// TIA Portal V20 export
FUNCTION_BLOCK "LER_AlignCalibration"   // FB100, LAD
// stored: Access Published, MemoryReserve 100, SetENOAutomatically false
   VAR_INPUT
      enable : Bool;
      Anode : Bool;
      Cathode : Bool;
      AxisXHomePos { ExternalAccessible := 'False'; ExternalVisible := 'False'; ExternalWritable := 'False'} : LReal;
      AxisY1HomePos { ExternalAccessible := 'False'; ExternalVisible := 'False'; ExternalWritable := 'False'} : LReal;
      AxisY2HomePos { ExternalAccessible := 'False'; ExternalVisible := 'False'; ExternalWritable := 'False'} : LReal;
   END_VAR
   VAR_OUTPUT
      Visiontrigger : Bool;
      error : Bool;
      busy : Bool;
      done : Bool;
      status : Word;
   END_VAR
   VAR_IN_OUT
      moduleInterface : "LER_typeAlignCalibrationInterface";
      AlignTableAxisX : DB_ANY;
      AlignTableAxisY1 : DB_ANY;
      AlignTableAxisY2 : DB_ANY;
   END_VAR
   VAR
      statAxisXMovePosition : Array[1..9] of LReal;
      statAxisY1MovePosition : Array[1..9] of LReal;
      statAxisY2MovePosition : Array[1..9] of LReal;
      instAlignTableAxisXMCMoveAbs : MC_MOVEABSOLUTE;
      instAlignTableAxisY1MCMoveAbs { S7_SetPoint := 'True'} : MC_MOVEABSOLUTE;
      instAlignTableAxisY2MCMoveAbs { S7_SetPoint := 'True'} : MC_MOVEABSOLUTE;
      statPulse { S7_SetPoint := 'True'} : Array[1..50] of Bool;
      statMoveXCmd : Array[1..10] of Bool;
      statMoveY1Cmd : Array[1..10] of Bool;
      statMoveY2Cmd : Array[1..10] of Bool;
      statVisionCmd : Array[1..10] of Bool;
      statTimer : Array[1..20] of TON_TIME;
      statAllMoveSeq : DInt;
      statManualMove : Bool;
   END_VAR
   VAR_TEMP
      tempAlignTableAxisX : REF_TO TO_SynchronousAxis;
      tempAlignTableAxisY1 : REF_TO TO_SynchronousAxis;
      tempAlignTableAxisY2 : REF_TO TO_SynchronousAxis;
   END_VAR
   VAR CONSTANT
      VISION_DELAY_TIME : Time := T#500ms;
   END_VAR
   VAR_TEMP   // added for the SCL form of the ladder/FBD networks
      _w1 : Bool;
      _w2 : Bool;
   END_VAR
BEGIN

REGION Network 1 (SCL): Axis Config
   #tempAlignTableAxisX ?= #AlignTableAxisX;
   #tempAlignTableAxisY1 ?= #AlignTableAxisY1;
   #tempAlignTableAxisY2 ?= #AlignTableAxisY2;
END_REGION

REGION Network 2: Standard Postion Config
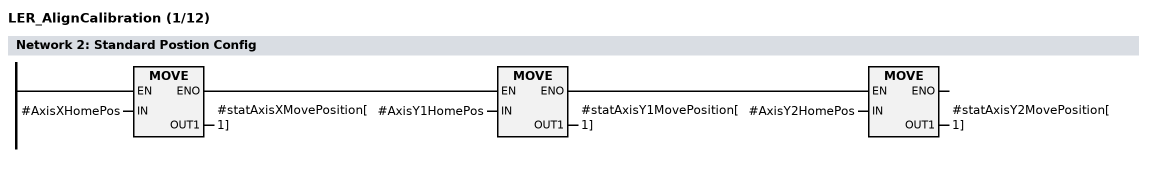
   RUNG wire#powerrail
      Move(in := #AxisXHomePos, out1 => #statAxisXMovePosition[1])
      Move(in := #AxisY1HomePos, out1 => #statAxisY1MovePosition[1])
      Move(in := #AxisY2HomePos, out1 => #statAxisY2MovePosition[1])
   END_RUNG
   // the same network as SCL:
   #statAxisXMovePosition[1] := #AxisXHomePos;
   #statAxisY1MovePosition[1] := #AxisY1HomePos;
   #statAxisY2MovePosition[1] := #AxisY2HomePos;
END_REGION

REGION Network 3: Anode MovePosition Config
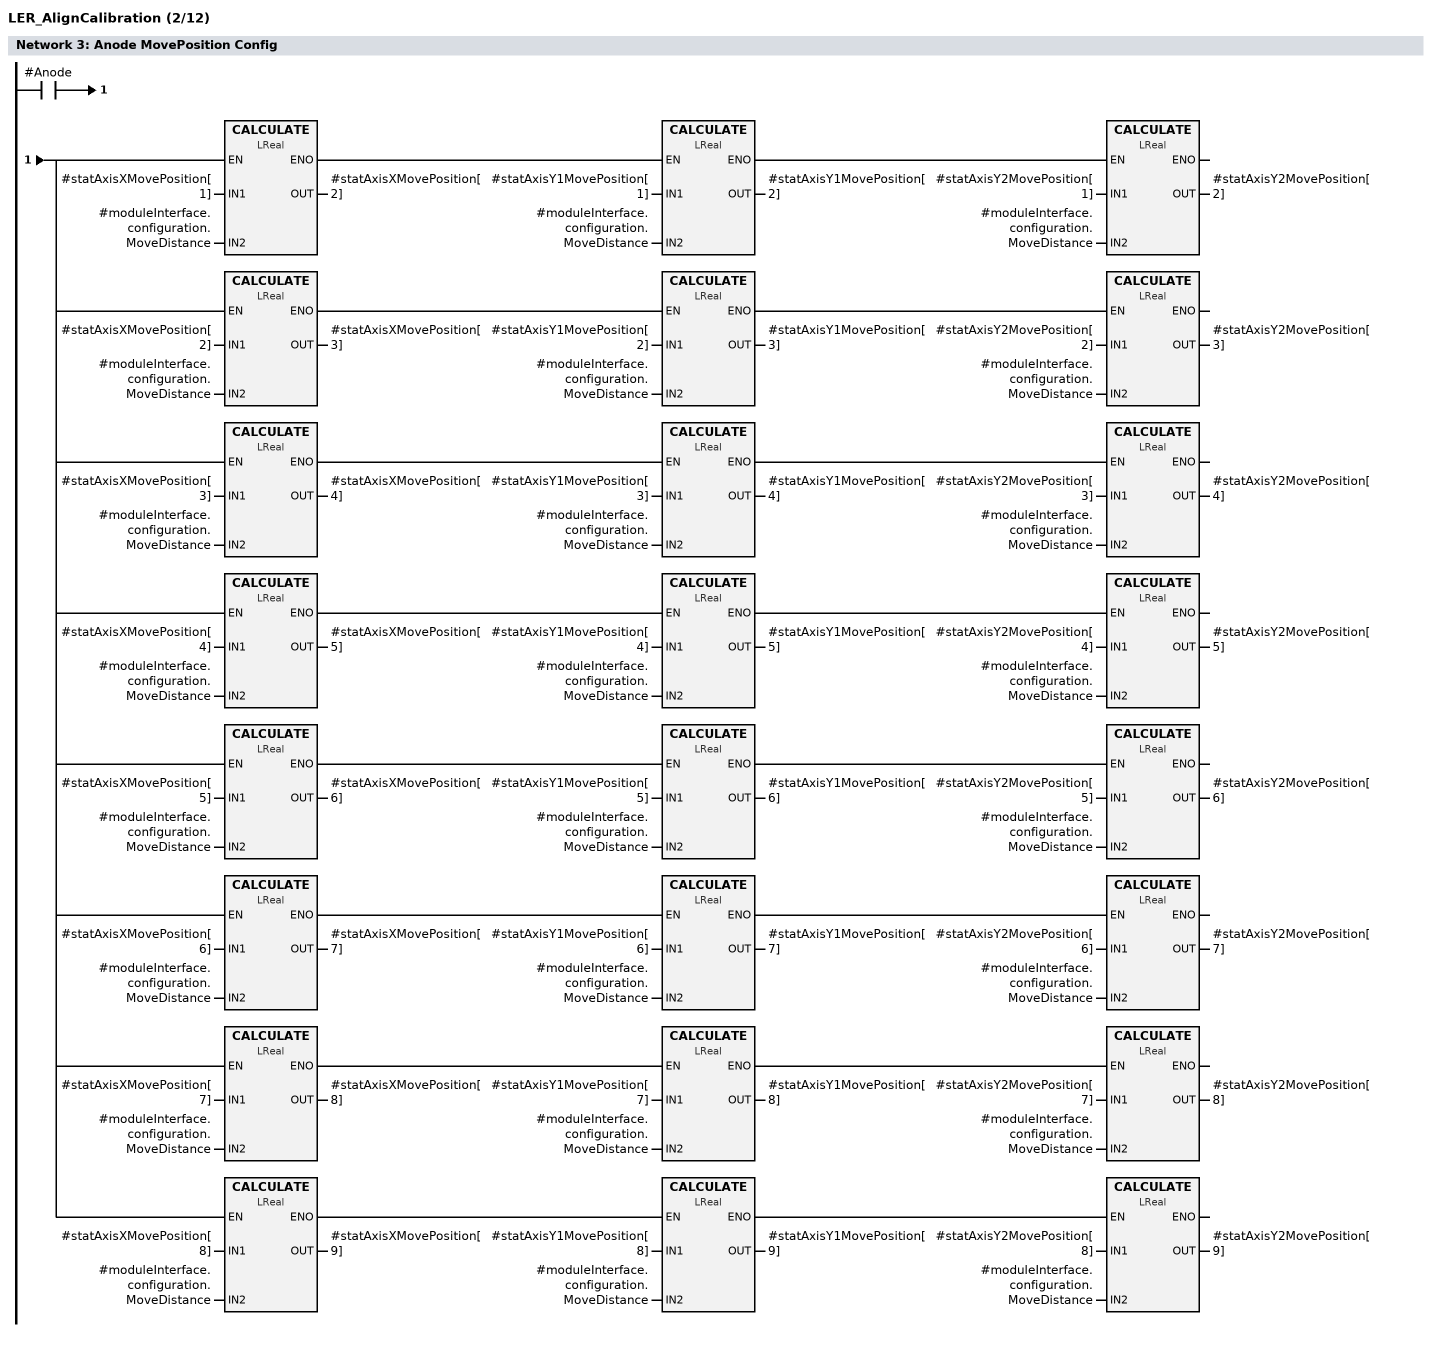
   RUNG wire#powerrail
      Contact( #Anode )
      wire#w1
      { S7_Templates := "SrcType := LReal"; S7_Expression := "IN1-IN2" } Calculate(in1 := #statAxisXMovePosition[1], in2 := #moduleInterface.configuration.MoveDistance, out => #statAxisXMovePosition[2])
      { S7_Templates := "SrcType := LReal"; S7_Expression := "IN1" } Calculate(in1 := #statAxisY1MovePosition[1], in2 := #moduleInterface.configuration.MoveDistance, out => #statAxisY1MovePosition[2])
      { S7_Templates := "SrcType := LReal"; S7_Expression := "IN1" } Calculate(in1 := #statAxisY2MovePosition[1], in2 := #moduleInterface.configuration.MoveDistance, out => #statAxisY2MovePosition[2])
   END_RUNG
   RUNG wire#w1
      { S7_Templates := "SrcType := LReal"; S7_Expression := "IN1" } Calculate(in1 := #statAxisXMovePosition[2], in2 := #moduleInterface.configuration.MoveDistance, out => #statAxisXMovePosition[3])
      { S7_Templates := "SrcType := LReal"; S7_Expression := "IN1+IN2" } Calculate(in1 := #statAxisY1MovePosition[2], in2 := #moduleInterface.configuration.MoveDistance, out => #statAxisY1MovePosition[3])
      { S7_Templates := "SrcType := LReal"; S7_Expression := "IN1-IN2" } Calculate(in1 := #statAxisY2MovePosition[2], in2 := #moduleInterface.configuration.MoveDistance, out => #statAxisY2MovePosition[3])
   END_RUNG
   RUNG wire#w1
      { S7_Templates := "SrcType := LReal"; S7_Expression := "IN1+IN2" } Calculate(in1 := #statAxisXMovePosition[3], in2 := #moduleInterface.configuration.MoveDistance, out => #statAxisXMovePosition[4])
      { S7_Templates := "SrcType := LReal"; S7_Expression := "IN1" } Calculate(in1 := #statAxisY1MovePosition[3], in2 := #moduleInterface.configuration.MoveDistance, out => #statAxisY1MovePosition[4])
      { S7_Templates := "SrcType := LReal"; S7_Expression := "IN1" } Calculate(in1 := #statAxisY2MovePosition[3], in2 := #moduleInterface.configuration.MoveDistance, out => #statAxisY2MovePosition[4])
   END_RUNG
   RUNG wire#w1
      { S7_Templates := "SrcType := LReal"; S7_Expression := "IN1+IN2" } Calculate(in1 := #statAxisXMovePosition[4], in2 := #moduleInterface.configuration.MoveDistance, out => #statAxisXMovePosition[5])
      { S7_Templates := "SrcType := LReal"; S7_Expression := "IN1" } Calculate(in1 := #statAxisY1MovePosition[4], in2 := #moduleInterface.configuration.MoveDistance, out => #statAxisY1MovePosition[5])
      { S7_Templates := "SrcType := LReal"; S7_Expression := "IN1" } Calculate(in1 := #statAxisY2MovePosition[4], in2 := #moduleInterface.configuration.MoveDistance, out => #statAxisY2MovePosition[5])
   END_RUNG
   RUNG wire#w1
      { S7_Templates := "SrcType := LReal"; S7_Expression := "IN1" } Calculate(in1 := #statAxisXMovePosition[5], in2 := #moduleInterface.configuration.MoveDistance, out => #statAxisXMovePosition[6])
      { S7_Templates := "SrcType := LReal"; S7_Expression := "IN1-IN2" } Calculate(in1 := #statAxisY1MovePosition[5], in2 := #moduleInterface.configuration.MoveDistance, out => #statAxisY1MovePosition[6])
      { S7_Templates := "SrcType := LReal"; S7_Expression := "IN1+IN2" } Calculate(in1 := #statAxisY2MovePosition[5], in2 := #moduleInterface.configuration.MoveDistance, out => #statAxisY2MovePosition[6])
   END_RUNG
   RUNG wire#w1
      { S7_Templates := "SrcType := LReal"; S7_Expression := "IN1" } Calculate(in1 := #statAxisXMovePosition[6], in2 := #moduleInterface.configuration.MoveDistance, out => #statAxisXMovePosition[7])
      { S7_Templates := "SrcType := LReal"; S7_Expression := "IN1-IN2" } Calculate(in1 := #statAxisY1MovePosition[6], in2 := #moduleInterface.configuration.MoveDistance, out => #statAxisY1MovePosition[7])
      { S7_Templates := "SrcType := LReal"; S7_Expression := "IN1+IN2" } Calculate(in1 := #statAxisY2MovePosition[6], in2 := #moduleInterface.configuration.MoveDistance, out => #statAxisY2MovePosition[7])
   END_RUNG
   RUNG wire#w1
      { S7_Templates := "SrcType := LReal"; S7_Expression := "IN1-IN2" } Calculate(in1 := #statAxisXMovePosition[7], in2 := #moduleInterface.configuration.MoveDistance, out => #statAxisXMovePosition[8])
      { S7_Templates := "SrcType := LReal"; S7_Expression := "IN1" } Calculate(in1 := #statAxisY1MovePosition[7], in2 := #moduleInterface.configuration.MoveDistance, out => #statAxisY1MovePosition[8])
      { S7_Templates := "SrcType := LReal"; S7_Expression := "IN1" } Calculate(in1 := #statAxisY2MovePosition[7], in2 := #moduleInterface.configuration.MoveDistance, out => #statAxisY2MovePosition[8])
   END_RUNG
   RUNG wire#w1
      { S7_Templates := "SrcType := LReal"; S7_Expression := "IN1-IN2" } Calculate(in1 := #statAxisXMovePosition[8], in2 := #moduleInterface.configuration.MoveDistance, out => #statAxisXMovePosition[9])
      { S7_Templates := "SrcType := LReal"; S7_Expression := "IN1" } Calculate(in1 := #statAxisY1MovePosition[8], in2 := #moduleInterface.configuration.MoveDistance, out => #statAxisY1MovePosition[9])
      { S7_Templates := "SrcType := LReal"; S7_Expression := "IN1" } Calculate(in1 := #statAxisY2MovePosition[8], in2 := #moduleInterface.configuration.MoveDistance, out => #statAxisY2MovePosition[9])
   END_RUNG
   // the same network as SCL:
   IF #Anode THEN
       #statAxisXMovePosition[2] := #statAxisXMovePosition[1]-#moduleInterface.configuration.MoveDistance;
       #statAxisY1MovePosition[2] := #statAxisY1MovePosition[1];
       #statAxisY2MovePosition[2] := #statAxisY2MovePosition[1];
       #statAxisXMovePosition[3] := #statAxisXMovePosition[2];
       #statAxisY1MovePosition[3] := #statAxisY1MovePosition[2]+#moduleInterface.configuration.MoveDistance;
       #statAxisY2MovePosition[3] := #statAxisY2MovePosition[2]-#moduleInterface.configuration.MoveDistance;
       #statAxisXMovePosition[4] := #statAxisXMovePosition[3]+#moduleInterface.configuration.MoveDistance;
       #statAxisY1MovePosition[4] := #statAxisY1MovePosition[3];
       #statAxisY2MovePosition[4] := #statAxisY2MovePosition[3];
       #statAxisXMovePosition[5] := #statAxisXMovePosition[4]+#moduleInterface.configuration.MoveDistance;
       #statAxisY1MovePosition[5] := #statAxisY1MovePosition[4];
       #statAxisY2MovePosition[5] := #statAxisY2MovePosition[4];
       #statAxisXMovePosition[6] := #statAxisXMovePosition[5];
       #statAxisY1MovePosition[6] := #statAxisY1MovePosition[5]-#moduleInterface.configuration.MoveDistance;
       #statAxisY2MovePosition[6] := #statAxisY2MovePosition[5]+#moduleInterface.configuration.MoveDistance;
       #statAxisXMovePosition[7] := #statAxisXMovePosition[6];
       #statAxisY1MovePosition[7] := #statAxisY1MovePosition[6]-#moduleInterface.configuration.MoveDistance;
       #statAxisY2MovePosition[7] := #statAxisY2MovePosition[6]+#moduleInterface.configuration.MoveDistance;
       #statAxisXMovePosition[8] := #statAxisXMovePosition[7]-#moduleInterface.configuration.MoveDistance;
       #statAxisY1MovePosition[8] := #statAxisY1MovePosition[7];
       #statAxisY2MovePosition[8] := #statAxisY2MovePosition[7];
       #statAxisXMovePosition[9] := #statAxisXMovePosition[8]-#moduleInterface.configuration.MoveDistance;
       #statAxisY1MovePosition[9] := #statAxisY1MovePosition[8];
       #statAxisY2MovePosition[9] := #statAxisY2MovePosition[8];
   END_IF;
END_REGION

REGION Network 4: Cathode MovePosition Config
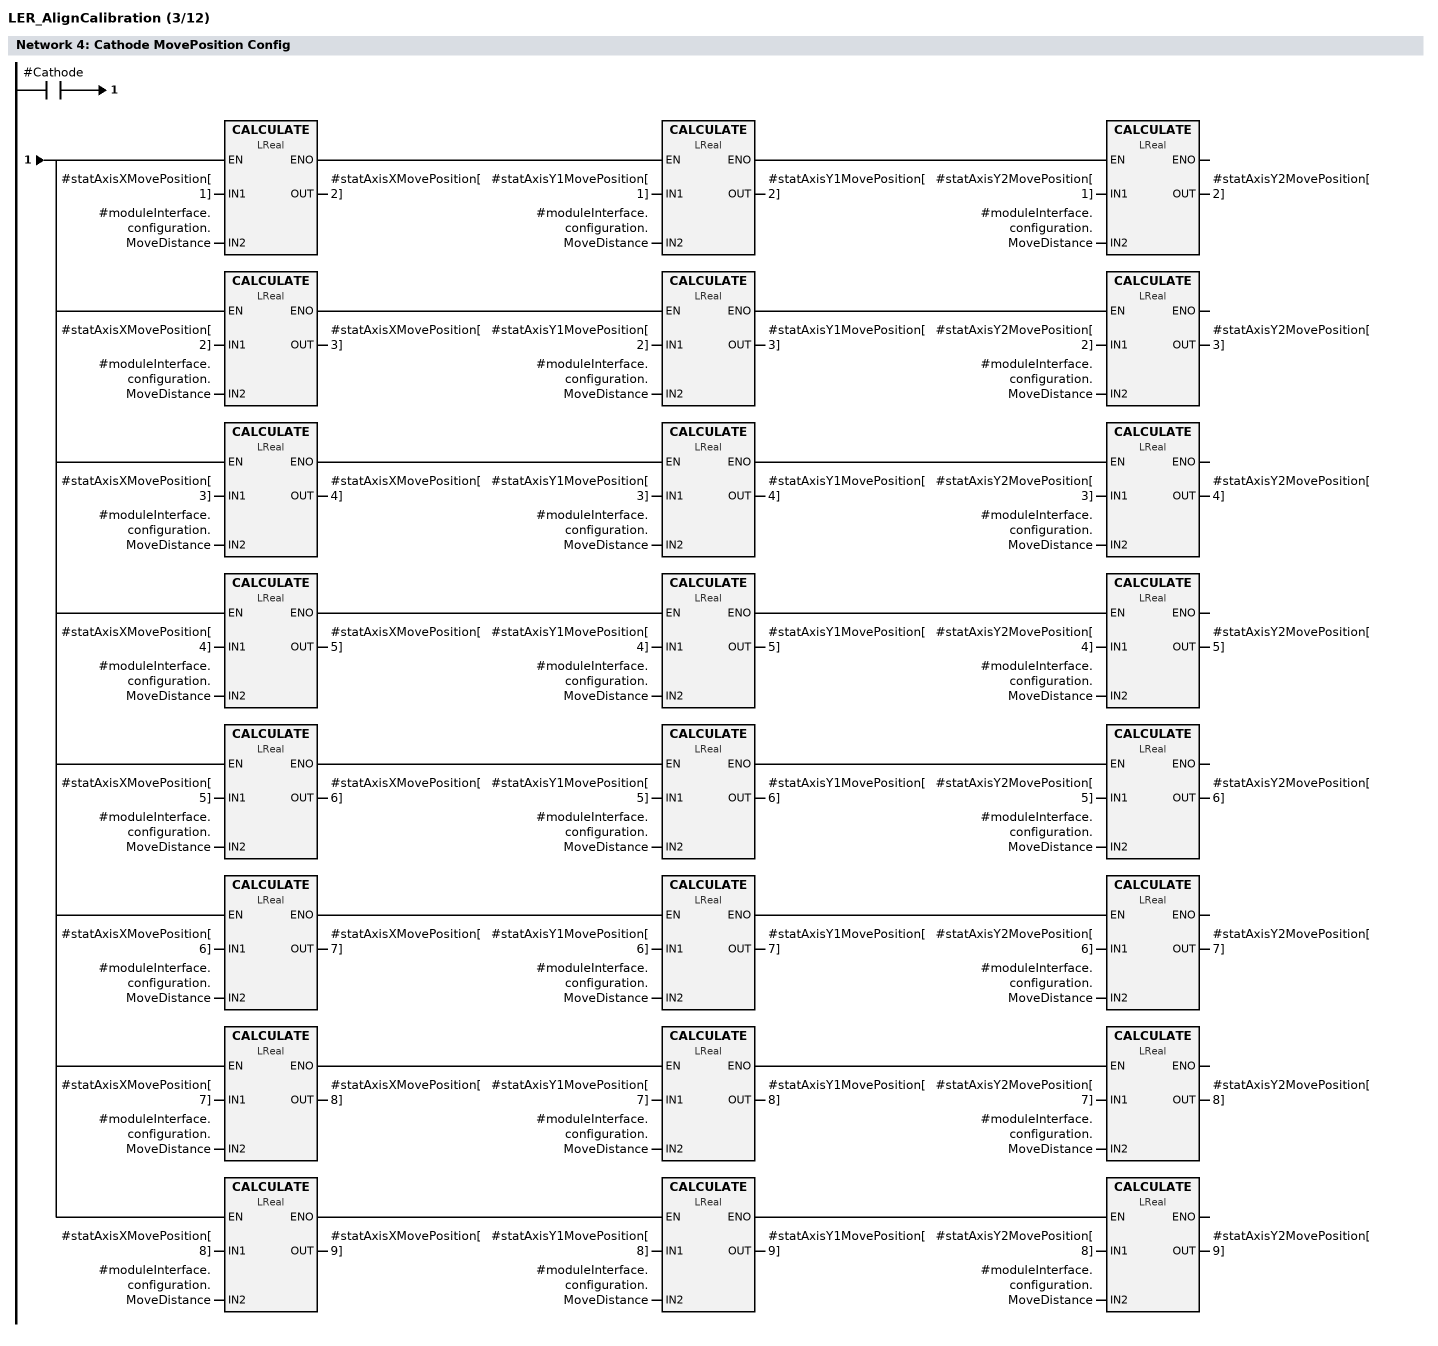
   RUNG wire#powerrail
      Contact( #Cathode )
      wire#w1
      { S7_Templates := "SrcType := LReal"; S7_Expression := "IN1+IN2" } Calculate(in1 := #statAxisXMovePosition[1], in2 := #moduleInterface.configuration.MoveDistance, out => #statAxisXMovePosition[2])
      { S7_Templates := "SrcType := LReal"; S7_Expression := "IN1" } Calculate(in1 := #statAxisY1MovePosition[1], in2 := #moduleInterface.configuration.MoveDistance, out => #statAxisY1MovePosition[2])
      { S7_Templates := "SrcType := LReal"; S7_Expression := "IN1" } Calculate(in1 := #statAxisY2MovePosition[1], in2 := #moduleInterface.configuration.MoveDistance, out => #statAxisY2MovePosition[2])
   END_RUNG
   RUNG wire#w1
      { S7_Templates := "SrcType := LReal"; S7_Expression := "IN1" } Calculate(in1 := #statAxisXMovePosition[2], in2 := #moduleInterface.configuration.MoveDistance, out => #statAxisXMovePosition[3])
      { S7_Templates := "SrcType := LReal"; S7_Expression := "IN1+IN2" } Calculate(in1 := #statAxisY1MovePosition[2], in2 := #moduleInterface.configuration.MoveDistance, out => #statAxisY1MovePosition[3])
      { S7_Templates := "SrcType := LReal"; S7_Expression := "IN1-IN2" } Calculate(in1 := #statAxisY2MovePosition[2], in2 := #moduleInterface.configuration.MoveDistance, out => #statAxisY2MovePosition[3])
   END_RUNG
   RUNG wire#w1
      { S7_Templates := "SrcType := LReal"; S7_Expression := "IN1-IN2" } Calculate(in1 := #statAxisXMovePosition[3], in2 := #moduleInterface.configuration.MoveDistance, out => #statAxisXMovePosition[4])
      { S7_Templates := "SrcType := LReal"; S7_Expression := "IN1" } Calculate(in1 := #statAxisY1MovePosition[3], in2 := #moduleInterface.configuration.MoveDistance, out => #statAxisY1MovePosition[4])
      { S7_Templates := "SrcType := LReal"; S7_Expression := "IN1" } Calculate(in1 := #statAxisY2MovePosition[3], in2 := #moduleInterface.configuration.MoveDistance, out => #statAxisY2MovePosition[4])
   END_RUNG
   RUNG wire#w1
      { S7_Templates := "SrcType := LReal"; S7_Expression := "IN1-IN2" } Calculate(in1 := #statAxisXMovePosition[4], in2 := #moduleInterface.configuration.MoveDistance, out => #statAxisXMovePosition[5])
      { S7_Templates := "SrcType := LReal"; S7_Expression := "IN1" } Calculate(in1 := #statAxisY1MovePosition[4], in2 := #moduleInterface.configuration.MoveDistance, out => #statAxisY1MovePosition[5])
      { S7_Templates := "SrcType := LReal"; S7_Expression := "IN1" } Calculate(in1 := #statAxisY2MovePosition[4], in2 := #moduleInterface.configuration.MoveDistance, out => #statAxisY2MovePosition[5])
   END_RUNG
   RUNG wire#w1
      { S7_Templates := "SrcType := LReal"; S7_Expression := "IN1" } Calculate(in1 := #statAxisXMovePosition[5], in2 := #moduleInterface.configuration.MoveDistance, out => #statAxisXMovePosition[6])
      { S7_Templates := "SrcType := LReal"; S7_Expression := "IN1-IN2" } Calculate(in1 := #statAxisY1MovePosition[5], in2 := #moduleInterface.configuration.MoveDistance, out => #statAxisY1MovePosition[6])
      { S7_Templates := "SrcType := LReal"; S7_Expression := "IN1+IN2" } Calculate(in1 := #statAxisY2MovePosition[5], in2 := #moduleInterface.configuration.MoveDistance, out => #statAxisY2MovePosition[6])
   END_RUNG
   RUNG wire#w1
      { S7_Templates := "SrcType := LReal"; S7_Expression := "IN1" } Calculate(in1 := #statAxisXMovePosition[6], in2 := #moduleInterface.configuration.MoveDistance, out => #statAxisXMovePosition[7])
      { S7_Templates := "SrcType := LReal"; S7_Expression := "IN1-IN2" } Calculate(in1 := #statAxisY1MovePosition[6], in2 := #moduleInterface.configuration.MoveDistance, out => #statAxisY1MovePosition[7])
      { S7_Templates := "SrcType := LReal"; S7_Expression := "IN1+IN2" } Calculate(in1 := #statAxisY2MovePosition[6], in2 := #moduleInterface.configuration.MoveDistance, out => #statAxisY2MovePosition[7])
   END_RUNG
   RUNG wire#w1
      { S7_Templates := "SrcType := LReal"; S7_Expression := "IN1+IN2" } Calculate(in1 := #statAxisXMovePosition[7], in2 := #moduleInterface.configuration.MoveDistance, out => #statAxisXMovePosition[8])
      { S7_Templates := "SrcType := LReal"; S7_Expression := "IN1" } Calculate(in1 := #statAxisY1MovePosition[7], in2 := #moduleInterface.configuration.MoveDistance, out => #statAxisY1MovePosition[8])
      { S7_Templates := "SrcType := LReal"; S7_Expression := "IN1" } Calculate(in1 := #statAxisY2MovePosition[7], in2 := #moduleInterface.configuration.MoveDistance, out => #statAxisY2MovePosition[8])
   END_RUNG
   RUNG wire#w1
      { S7_Templates := "SrcType := LReal"; S7_Expression := "IN1+IN2" } Calculate(in1 := #statAxisXMovePosition[8], in2 := #moduleInterface.configuration.MoveDistance, out => #statAxisXMovePosition[9])
      { S7_Templates := "SrcType := LReal"; S7_Expression := "IN1" } Calculate(in1 := #statAxisY1MovePosition[8], in2 := #moduleInterface.configuration.MoveDistance, out => #statAxisY1MovePosition[9])
      { S7_Templates := "SrcType := LReal"; S7_Expression := "IN1" } Calculate(in1 := #statAxisY2MovePosition[8], in2 := #moduleInterface.configuration.MoveDistance, out => #statAxisY2MovePosition[9])
   END_RUNG
   // the same network as SCL:
   IF #Cathode THEN
       #statAxisXMovePosition[2] := #statAxisXMovePosition[1]+#moduleInterface.configuration.MoveDistance;
       #statAxisY1MovePosition[2] := #statAxisY1MovePosition[1];
       #statAxisY2MovePosition[2] := #statAxisY2MovePosition[1];
       #statAxisXMovePosition[3] := #statAxisXMovePosition[2];
       #statAxisY1MovePosition[3] := #statAxisY1MovePosition[2]+#moduleInterface.configuration.MoveDistance;
       #statAxisY2MovePosition[3] := #statAxisY2MovePosition[2]-#moduleInterface.configuration.MoveDistance;
       #statAxisXMovePosition[4] := #statAxisXMovePosition[3]-#moduleInterface.configuration.MoveDistance;
       #statAxisY1MovePosition[4] := #statAxisY1MovePosition[3];
       #statAxisY2MovePosition[4] := #statAxisY2MovePosition[3];
       #statAxisXMovePosition[5] := #statAxisXMovePosition[4]-#moduleInterface.configuration.MoveDistance;
       #statAxisY1MovePosition[5] := #statAxisY1MovePosition[4];
       #statAxisY2MovePosition[5] := #statAxisY2MovePosition[4];
       #statAxisXMovePosition[6] := #statAxisXMovePosition[5];
       #statAxisY1MovePosition[6] := #statAxisY1MovePosition[5]-#moduleInterface.configuration.MoveDistance;
       #statAxisY2MovePosition[6] := #statAxisY2MovePosition[5]+#moduleInterface.configuration.MoveDistance;
       #statAxisXMovePosition[7] := #statAxisXMovePosition[6];
       #statAxisY1MovePosition[7] := #statAxisY1MovePosition[6]-#moduleInterface.configuration.MoveDistance;
       #statAxisY2MovePosition[7] := #statAxisY2MovePosition[6]+#moduleInterface.configuration.MoveDistance;
       #statAxisXMovePosition[8] := #statAxisXMovePosition[7]+#moduleInterface.configuration.MoveDistance;
       #statAxisY1MovePosition[8] := #statAxisY1MovePosition[7];
       #statAxisY2MovePosition[8] := #statAxisY2MovePosition[7];
       #statAxisXMovePosition[9] := #statAxisXMovePosition[8]+#moduleInterface.configuration.MoveDistance;
       #statAxisY1MovePosition[9] := #statAxisY1MovePosition[8];
       #statAxisY2MovePosition[9] := #statAxisY2MovePosition[8];
   END_IF;
END_REGION

REGION Network 5: All Move Seq Start/Stop And Error Check
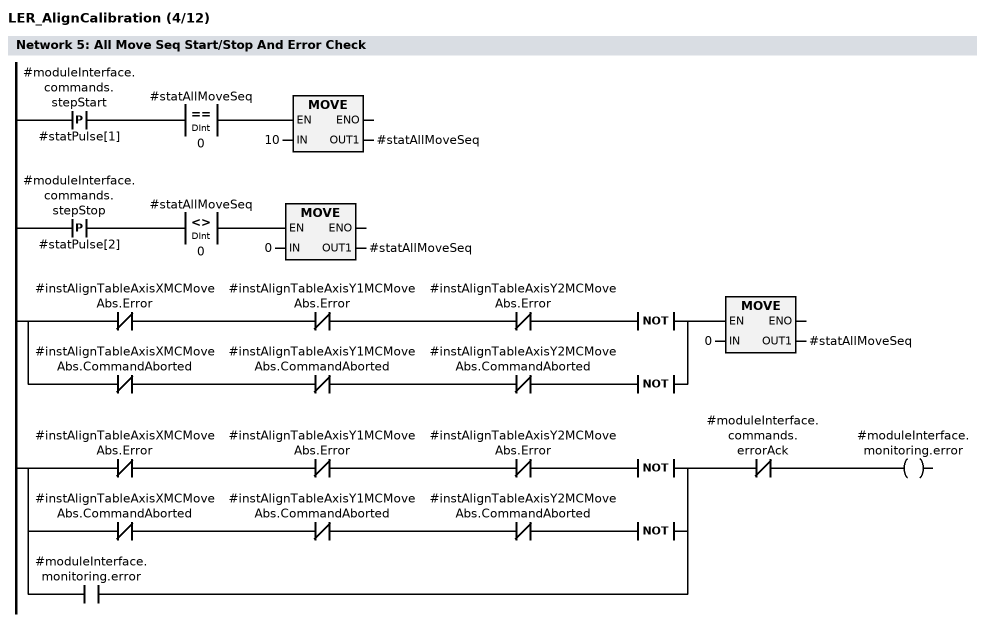
   RUNG wire#powerrail
      P_Contact(operand := #moduleInterface.commands.stepStart, bit := #statPulse[1])
      { S7_Templates := "SrcType := DInt" } EQ_Contact(in1 := #statAllMoveSeq, in2 := 0)
      Move(in := 10, out1 => #statAllMoveSeq)
   END_RUNG
   RUNG wire#powerrail
      P_Contact(operand := #moduleInterface.commands.stepStop, bit := #statPulse[2])
      { S7_Templates := "SrcType := DInt" } NE_Contact(in1 := #statAllMoveSeq, in2 := 0)
      Move(in := 0, out1 => #statAllMoveSeq)
   END_RUNG
   RUNG wire#powerrail
      I_Contact( #instAlignTableAxisXMCMoveAbs.Error )
      I_Contact( #instAlignTableAxisY1MCMoveAbs.Error )
      I_Contact( #instAlignTableAxisY2MCMoveAbs.Error )
      Not()
      wire#w1
      Move(in := 0, out1 => #statAllMoveSeq)
   END_RUNG
   RUNG wire#powerrail
      I_Contact( #instAlignTableAxisXMCMoveAbs.CommandAborted )
      I_Contact( #instAlignTableAxisY1MCMoveAbs.CommandAborted )
      I_Contact( #instAlignTableAxisY2MCMoveAbs.CommandAborted )
      Not()
   END_RUNG wire#w1
   RUNG wire#powerrail
      I_Contact( #instAlignTableAxisXMCMoveAbs.Error )
      I_Contact( #instAlignTableAxisY1MCMoveAbs.Error )
      I_Contact( #instAlignTableAxisY2MCMoveAbs.Error )
      Not()
      wire#w2
      I_Contact( #moduleInterface.commands.errorAck )
      Coil( #moduleInterface.monitoring.error )
   END_RUNG
   RUNG wire#powerrail
      I_Contact( #instAlignTableAxisXMCMoveAbs.CommandAborted )
      I_Contact( #instAlignTableAxisY1MCMoveAbs.CommandAborted )
      I_Contact( #instAlignTableAxisY2MCMoveAbs.CommandAborted )
      Not()
   END_RUNG wire#w2
   RUNG wire#powerrail
      Contact( #moduleInterface.monitoring.error )
   END_RUNG wire#w2
   // the same network as SCL:
   #_w1 := #moduleInterface.commands.stepStart AND NOT #statPulse[1];   // rising edge of #moduleInterface.commands.stepStart
   #statPulse[1] := #moduleInterface.commands.stepStart;
   IF #_w1 AND (#statAllMoveSeq = 0) THEN #statAllMoveSeq := 10; END_IF;
   #_w2 := #moduleInterface.commands.stepStop AND NOT #statPulse[2];   // rising edge of #moduleInterface.commands.stepStop
   #statPulse[2] := #moduleInterface.commands.stepStop;
   IF #_w2 AND (#statAllMoveSeq <> 0) THEN #statAllMoveSeq := 0; END_IF;
   IF NOT (NOT #instAlignTableAxisXMCMoveAbs.Error AND NOT #instAlignTableAxisY1MCMoveAbs.Error AND NOT #instAlignTableAxisY2MCMoveAbs.Error) OR NOT (NOT #instAlignTableAxisXMCMoveAbs.CommandAborted AND NOT #instAlignTableAxisY1MCMoveAbs.CommandAborted AND NOT #instAlignTableAxisY2MCMoveAbs.CommandAborted) THEN
       #statAllMoveSeq := 0;
   END_IF;
   #moduleInterface.monitoring.error := (NOT (NOT #instAlignTableAxisXMCMoveAbs.Error AND NOT #instAlignTableAxisY1MCMoveAbs.Error AND NOT #instAlignTableAxisY2MCMoveAbs.Error) OR NOT (NOT #instAlignTableAxisXMCMoveAbs.CommandAborted AND NOT #instAlignTableAxisY1MCMoveAbs.CommandAborted AND NOT #instAlignTableAxisY2MCMoveAbs.CommandAborted) OR #moduleInterface.monitoring.error) AND NOT #moduleInterface.commands.errorAck;
END_REGION

REGION Network 6: Manual Move Pos Check
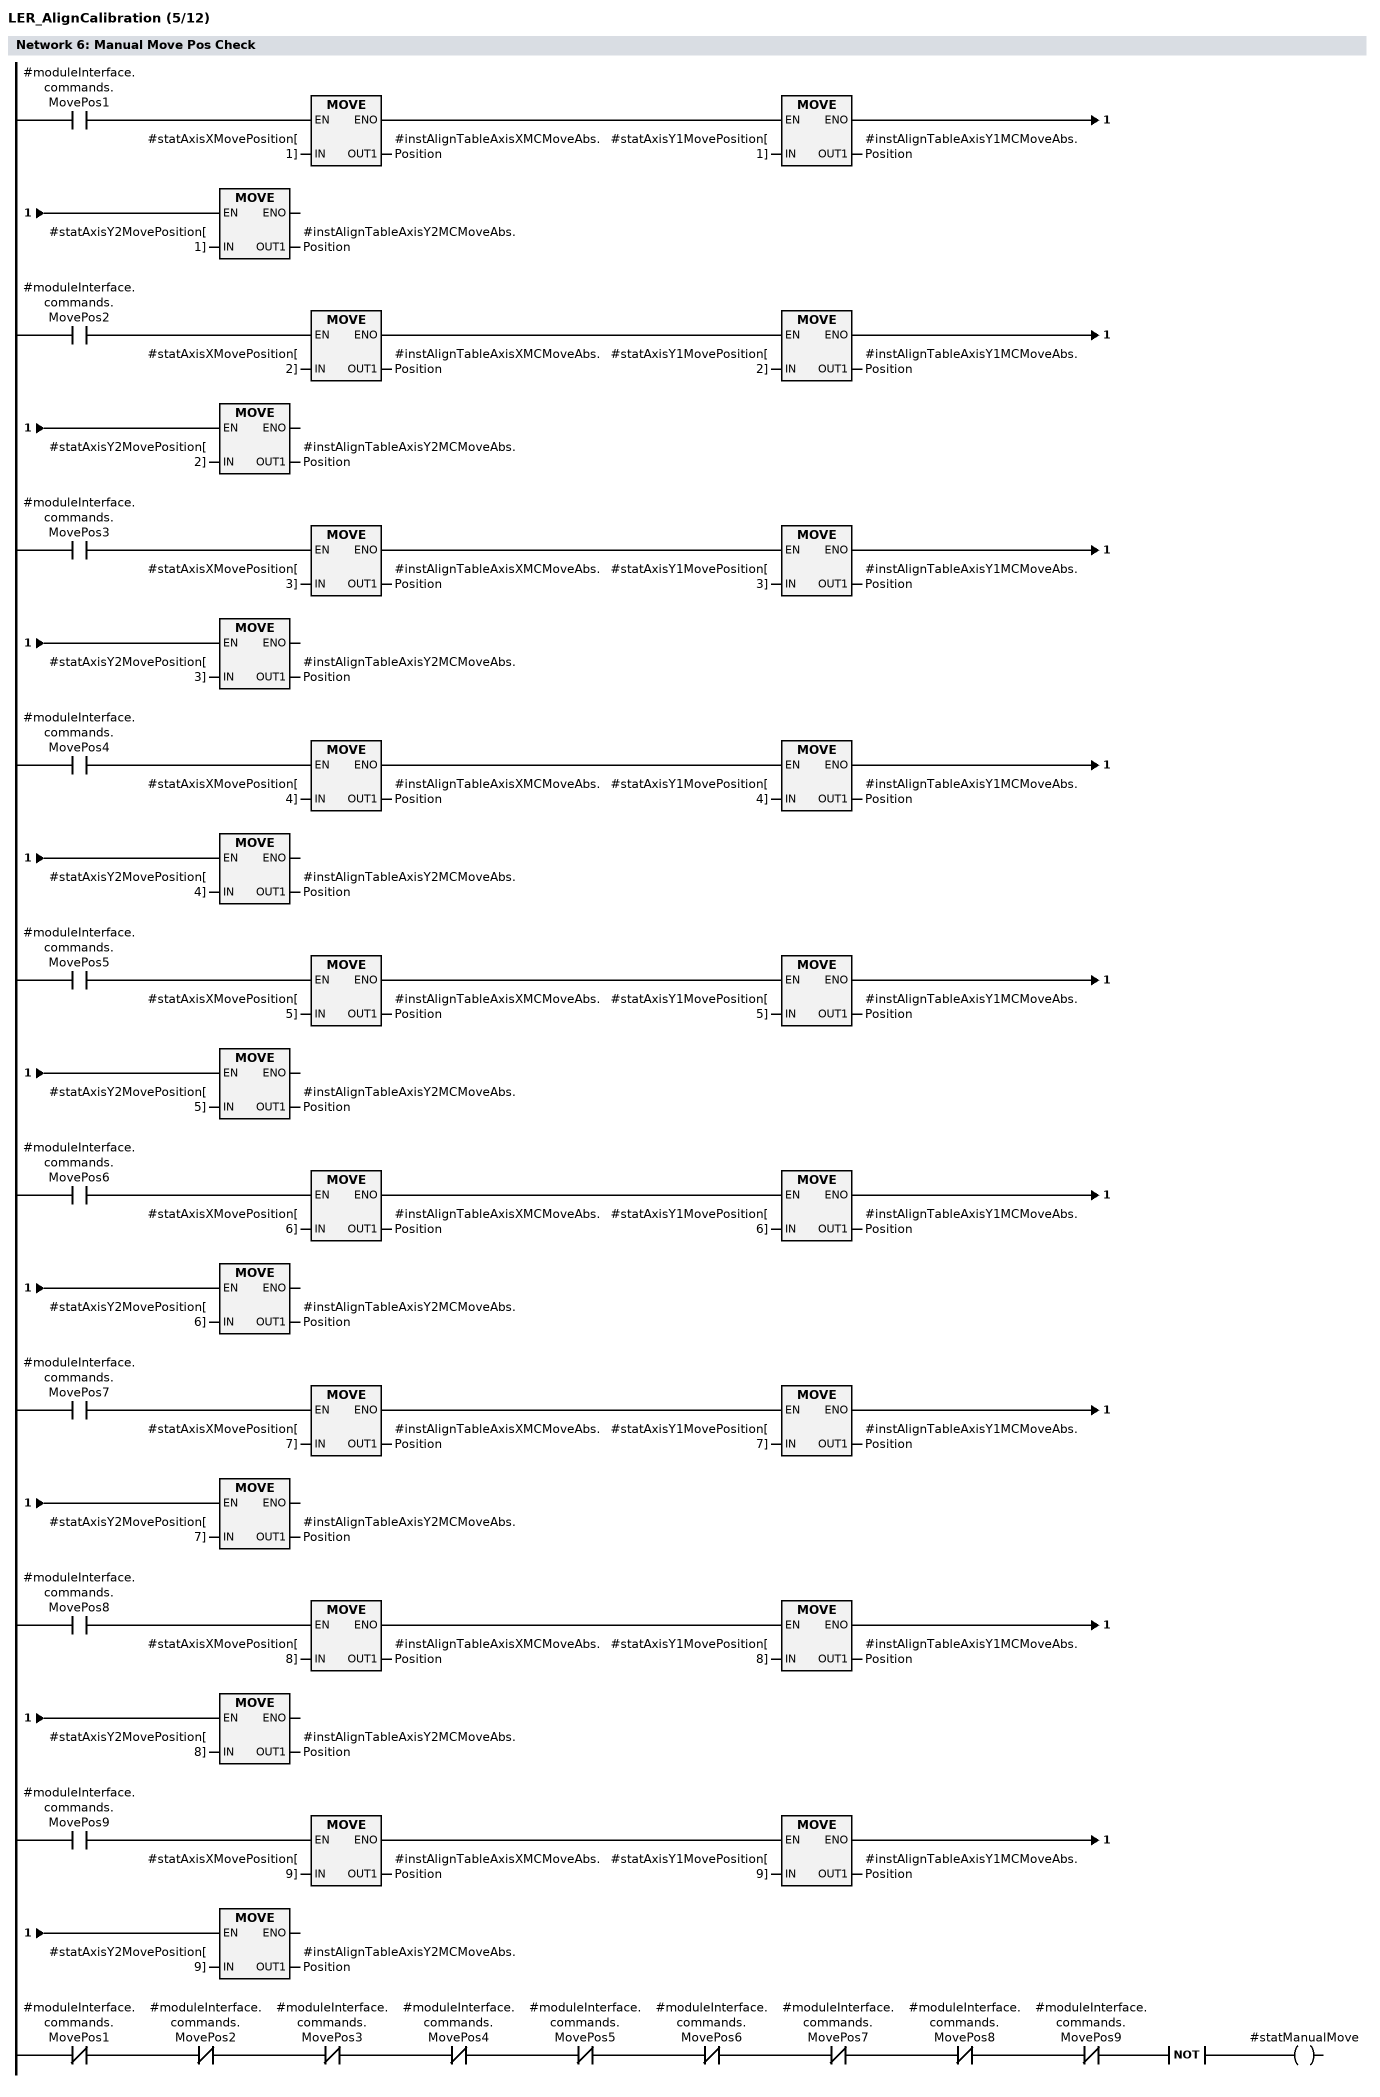
   RUNG wire#powerrail
      Contact( #moduleInterface.commands.MovePos1 )
      Move(in := #statAxisXMovePosition[1], out1 => #instAlignTableAxisXMCMoveAbs.Position)
      Move(in := #statAxisY1MovePosition[1], out1 => #instAlignTableAxisY1MCMoveAbs.Position)
      Move(in := #statAxisY2MovePosition[1], out1 => #instAlignTableAxisY2MCMoveAbs.Position)
   END_RUNG
   RUNG wire#powerrail
      Contact( #moduleInterface.commands.MovePos2 )
      Move(in := #statAxisXMovePosition[2], out1 => #instAlignTableAxisXMCMoveAbs.Position)
      Move(in := #statAxisY1MovePosition[2], out1 => #instAlignTableAxisY1MCMoveAbs.Position)
      Move(in := #statAxisY2MovePosition[2], out1 => #instAlignTableAxisY2MCMoveAbs.Position)
   END_RUNG
   RUNG wire#powerrail
      Contact( #moduleInterface.commands.MovePos3 )
      Move(in := #statAxisXMovePosition[3], out1 => #instAlignTableAxisXMCMoveAbs.Position)
      Move(in := #statAxisY1MovePosition[3], out1 => #instAlignTableAxisY1MCMoveAbs.Position)
      Move(in := #statAxisY2MovePosition[3], out1 => #instAlignTableAxisY2MCMoveAbs.Position)
   END_RUNG
   RUNG wire#powerrail
      Contact( #moduleInterface.commands.MovePos4 )
      Move(in := #statAxisXMovePosition[4], out1 => #instAlignTableAxisXMCMoveAbs.Position)
      Move(in := #statAxisY1MovePosition[4], out1 => #instAlignTableAxisY1MCMoveAbs.Position)
      Move(in := #statAxisY2MovePosition[4], out1 => #instAlignTableAxisY2MCMoveAbs.Position)
   END_RUNG
   RUNG wire#powerrail
      Contact( #moduleInterface.commands.MovePos5 )
      Move(in := #statAxisXMovePosition[5], out1 => #instAlignTableAxisXMCMoveAbs.Position)
      Move(in := #statAxisY1MovePosition[5], out1 => #instAlignTableAxisY1MCMoveAbs.Position)
      Move(in := #statAxisY2MovePosition[5], out1 => #instAlignTableAxisY2MCMoveAbs.Position)
   END_RUNG
   RUNG wire#powerrail
      Contact( #moduleInterface.commands.MovePos6 )
      Move(in := #statAxisXMovePosition[6], out1 => #instAlignTableAxisXMCMoveAbs.Position)
      Move(in := #statAxisY1MovePosition[6], out1 => #instAlignTableAxisY1MCMoveAbs.Position)
      Move(in := #statAxisY2MovePosition[6], out1 => #instAlignTableAxisY2MCMoveAbs.Position)
   END_RUNG
   RUNG wire#powerrail
      Contact( #moduleInterface.commands.MovePos7 )
      Move(in := #statAxisXMovePosition[7], out1 => #instAlignTableAxisXMCMoveAbs.Position)
      Move(in := #statAxisY1MovePosition[7], out1 => #instAlignTableAxisY1MCMoveAbs.Position)
      Move(in := #statAxisY2MovePosition[7], out1 => #instAlignTableAxisY2MCMoveAbs.Position)
   END_RUNG
   RUNG wire#powerrail
      Contact( #moduleInterface.commands.MovePos8 )
      Move(in := #statAxisXMovePosition[8], out1 => #instAlignTableAxisXMCMoveAbs.Position)
      Move(in := #statAxisY1MovePosition[8], out1 => #instAlignTableAxisY1MCMoveAbs.Position)
      Move(in := #statAxisY2MovePosition[8], out1 => #instAlignTableAxisY2MCMoveAbs.Position)
   END_RUNG
   RUNG wire#powerrail
      Contact( #moduleInterface.commands.MovePos9 )
      Move(in := #statAxisXMovePosition[9], out1 => #instAlignTableAxisXMCMoveAbs.Position)
      Move(in := #statAxisY1MovePosition[9], out1 => #instAlignTableAxisY1MCMoveAbs.Position)
      Move(in := #statAxisY2MovePosition[9], out1 => #instAlignTableAxisY2MCMoveAbs.Position)
   END_RUNG
   RUNG wire#powerrail
      I_Contact( #moduleInterface.commands.MovePos1 )
      I_Contact( #moduleInterface.commands.MovePos2 )
      I_Contact( #moduleInterface.commands.MovePos3 )
      I_Contact( #moduleInterface.commands.MovePos4 )
      I_Contact( #moduleInterface.commands.MovePos5 )
      I_Contact( #moduleInterface.commands.MovePos6 )
      I_Contact( #moduleInterface.commands.MovePos7 )
      I_Contact( #moduleInterface.commands.MovePos8 )
      I_Contact( #moduleInterface.commands.MovePos9 )
      Not()
      Coil( #statManualMove )
   END_RUNG
   // the same network as SCL:
   IF #moduleInterface.commands.MovePos1 THEN
       #instAlignTableAxisXMCMoveAbs.Position := #statAxisXMovePosition[1];
       #instAlignTableAxisY1MCMoveAbs.Position := #statAxisY1MovePosition[1];
       #instAlignTableAxisY2MCMoveAbs.Position := #statAxisY2MovePosition[1];
   END_IF;
   IF #moduleInterface.commands.MovePos2 THEN
       #instAlignTableAxisXMCMoveAbs.Position := #statAxisXMovePosition[2];
       #instAlignTableAxisY1MCMoveAbs.Position := #statAxisY1MovePosition[2];
       #instAlignTableAxisY2MCMoveAbs.Position := #statAxisY2MovePosition[2];
   END_IF;
   IF #moduleInterface.commands.MovePos3 THEN
       #instAlignTableAxisXMCMoveAbs.Position := #statAxisXMovePosition[3];
       #instAlignTableAxisY1MCMoveAbs.Position := #statAxisY1MovePosition[3];
       #instAlignTableAxisY2MCMoveAbs.Position := #statAxisY2MovePosition[3];
   END_IF;
   IF #moduleInterface.commands.MovePos4 THEN
       #instAlignTableAxisXMCMoveAbs.Position := #statAxisXMovePosition[4];
       #instAlignTableAxisY1MCMoveAbs.Position := #statAxisY1MovePosition[4];
       #instAlignTableAxisY2MCMoveAbs.Position := #statAxisY2MovePosition[4];
   END_IF;
   IF #moduleInterface.commands.MovePos5 THEN
       #instAlignTableAxisXMCMoveAbs.Position := #statAxisXMovePosition[5];
       #instAlignTableAxisY1MCMoveAbs.Position := #statAxisY1MovePosition[5];
       #instAlignTableAxisY2MCMoveAbs.Position := #statAxisY2MovePosition[5];
   END_IF;
   IF #moduleInterface.commands.MovePos6 THEN
       #instAlignTableAxisXMCMoveAbs.Position := #statAxisXMovePosition[6];
       #instAlignTableAxisY1MCMoveAbs.Position := #statAxisY1MovePosition[6];
       #instAlignTableAxisY2MCMoveAbs.Position := #statAxisY2MovePosition[6];
   END_IF;
   IF #moduleInterface.commands.MovePos7 THEN
       #instAlignTableAxisXMCMoveAbs.Position := #statAxisXMovePosition[7];
       #instAlignTableAxisY1MCMoveAbs.Position := #statAxisY1MovePosition[7];
       #instAlignTableAxisY2MCMoveAbs.Position := #statAxisY2MovePosition[7];
   END_IF;
   IF #moduleInterface.commands.MovePos8 THEN
       #instAlignTableAxisXMCMoveAbs.Position := #statAxisXMovePosition[8];
       #instAlignTableAxisY1MCMoveAbs.Position := #statAxisY1MovePosition[8];
       #instAlignTableAxisY2MCMoveAbs.Position := #statAxisY2MovePosition[8];
   END_IF;
   IF #moduleInterface.commands.MovePos9 THEN
       #instAlignTableAxisXMCMoveAbs.Position := #statAxisXMovePosition[9];
       #instAlignTableAxisY1MCMoveAbs.Position := #statAxisY1MovePosition[9];
       #instAlignTableAxisY2MCMoveAbs.Position := #statAxisY2MovePosition[9];
   END_IF;
   #statManualMove := NOT (NOT #moduleInterface.commands.MovePos1 AND NOT #moduleInterface.commands.MovePos2 AND NOT #moduleInterface.commands.MovePos3 AND NOT #moduleInterface.commands.MovePos4 AND NOT #moduleInterface.commands.MovePos5 AND NOT #moduleInterface.commands.MovePos6 AND NOT #moduleInterface.commands.MovePos7 AND NOT #moduleInterface.commands.MovePos8 AND NOT #moduleInterface.commands.MovePos9);
END_REGION

REGION Network 7: === Sequence Start ===
END_REGION

REGION Network 8: All Move Seq Pos 1 [Seq 10]
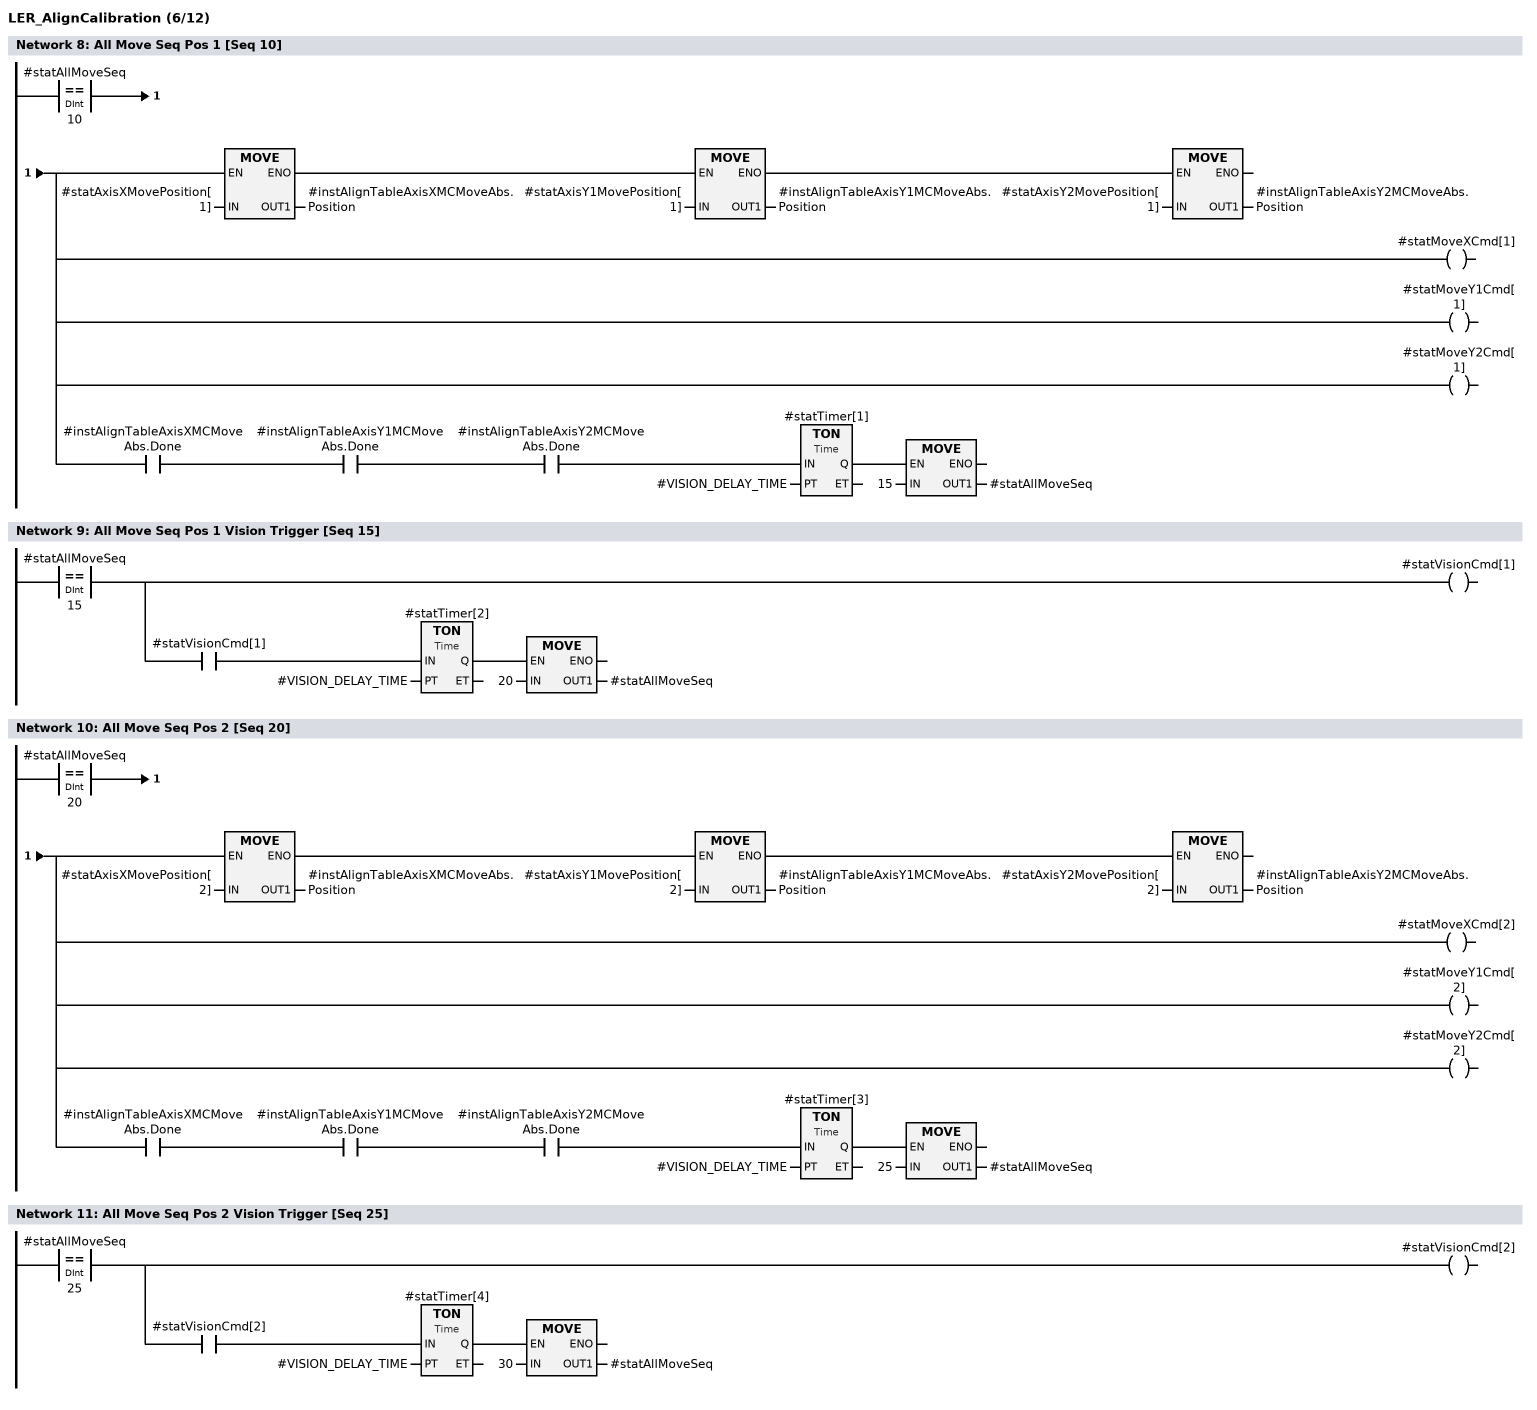
   RUNG wire#powerrail
      { S7_Templates := "SrcType := DInt" } EQ_Contact(in1 := #statAllMoveSeq, in2 := 10)
      wire#w1
      Move(in := #statAxisXMovePosition[1], out1 => #instAlignTableAxisXMCMoveAbs.Position)
      Move(in := #statAxisY1MovePosition[1], out1 => #instAlignTableAxisY1MCMoveAbs.Position)
      Move(in := #statAxisY2MovePosition[1], out1 => #instAlignTableAxisY2MCMoveAbs.Position)
   END_RUNG
   RUNG wire#w1
      Coil( #statMoveXCmd[1] )
   END_RUNG
   RUNG wire#w1
      Coil( #statMoveY1Cmd[1] )
   END_RUNG
   RUNG wire#w1
      Coil( #statMoveY2Cmd[1] )
   END_RUNG
   RUNG wire#w1
      Contact( #instAlignTableAxisXMCMoveAbs.Done )
      Contact( #instAlignTableAxisY1MCMoveAbs.Done )
      Contact( #instAlignTableAxisY2MCMoveAbs.Done )
      { S7_Templates := "time_type := Time" } #statTimer[1].TON(pt := #VISION_DELAY_TIME, et =>)
      Move(in := 15, out1 => #statAllMoveSeq)
   END_RUNG
   // the same network as SCL:
   #_w1 := #statAllMoveSeq = 10;
   IF #_w1 THEN
       #instAlignTableAxisXMCMoveAbs.Position := #statAxisXMovePosition[1];
       #instAlignTableAxisY1MCMoveAbs.Position := #statAxisY1MovePosition[1];
       #instAlignTableAxisY2MCMoveAbs.Position := #statAxisY2MovePosition[1];
   END_IF;
   #statMoveXCmd[1] := #_w1;
   #statMoveY1Cmd[1] := #_w1;
   #statMoveY2Cmd[1] := #_w1;
   #statTimer[1].TON(IN := #_w1 AND #instAlignTableAxisXMCMoveAbs.Done AND #instAlignTableAxisY1MCMoveAbs.Done AND #instAlignTableAxisY2MCMoveAbs.Done,
                     PT := #VISION_DELAY_TIME);
   IF #statTimer[1].Q THEN #statAllMoveSeq := 15; END_IF;
END_REGION

REGION Network 9: All Move Seq Pos 1 Vision Trigger [Seq 15]
   RUNG wire#powerrail
      { S7_Templates := "SrcType := DInt" } EQ_Contact(in1 := #statAllMoveSeq, in2 := 15)
      wire#w1
      Coil( #statVisionCmd[1] )
   END_RUNG
   RUNG wire#w1
      Contact( #statVisionCmd[1] )
      { S7_Templates := "time_type := Time" } #statTimer[2].TON(pt := #VISION_DELAY_TIME, et =>)
      Move(in := 20, out1 => #statAllMoveSeq)
   END_RUNG
   // the same network as SCL:
   #statVisionCmd[1] := #statAllMoveSeq = 15;
   #statTimer[2].TON(IN := (#statAllMoveSeq = 15) AND #statVisionCmd[1], PT := #VISION_DELAY_TIME);
   IF #statTimer[2].Q THEN #statAllMoveSeq := 20; END_IF;
END_REGION

REGION Network 10: All Move Seq Pos 2 [Seq 20]
   RUNG wire#powerrail
      { S7_Templates := "SrcType := DInt" } EQ_Contact(in1 := #statAllMoveSeq, in2 := 20)
      wire#w1
      Move(in := #statAxisXMovePosition[2], out1 => #instAlignTableAxisXMCMoveAbs.Position)
      Move(in := #statAxisY1MovePosition[2], out1 => #instAlignTableAxisY1MCMoveAbs.Position)
      Move(in := #statAxisY2MovePosition[2], out1 => #instAlignTableAxisY2MCMoveAbs.Position)
   END_RUNG
   RUNG wire#w1
      Coil( #statMoveXCmd[2] )
   END_RUNG
   RUNG wire#w1
      Coil( #statMoveY1Cmd[2] )
   END_RUNG
   RUNG wire#w1
      Coil( #statMoveY2Cmd[2] )
   END_RUNG
   RUNG wire#w1
      Contact( #instAlignTableAxisXMCMoveAbs.Done )
      Contact( #instAlignTableAxisY1MCMoveAbs.Done )
      Contact( #instAlignTableAxisY2MCMoveAbs.Done )
      { S7_Templates := "time_type := Time" } #statTimer[3].TON(pt := #VISION_DELAY_TIME, et =>)
      Move(in := 25, out1 => #statAllMoveSeq)
   END_RUNG
   // the same network as SCL:
   #_w1 := #statAllMoveSeq = 20;
   IF #_w1 THEN
       #instAlignTableAxisXMCMoveAbs.Position := #statAxisXMovePosition[2];
       #instAlignTableAxisY1MCMoveAbs.Position := #statAxisY1MovePosition[2];
       #instAlignTableAxisY2MCMoveAbs.Position := #statAxisY2MovePosition[2];
   END_IF;
   #statMoveXCmd[2] := #_w1;
   #statMoveY1Cmd[2] := #_w1;
   #statMoveY2Cmd[2] := #_w1;
   #statTimer[3].TON(IN := #_w1 AND #instAlignTableAxisXMCMoveAbs.Done AND #instAlignTableAxisY1MCMoveAbs.Done AND #instAlignTableAxisY2MCMoveAbs.Done,
                     PT := #VISION_DELAY_TIME);
   IF #statTimer[3].Q THEN #statAllMoveSeq := 25; END_IF;
END_REGION

REGION Network 11: All Move Seq Pos 2 Vision Trigger [Seq 25]
   RUNG wire#powerrail
      { S7_Templates := "SrcType := DInt" } EQ_Contact(in1 := #statAllMoveSeq, in2 := 25)
      wire#w1
      Coil( #statVisionCmd[2] )
   END_RUNG
   RUNG wire#w1
      Contact( #statVisionCmd[2] )
      { S7_Templates := "time_type := Time" } #statTimer[4].TON(pt := #VISION_DELAY_TIME, et =>)
      Move(in := 30, out1 => #statAllMoveSeq)
   END_RUNG
   // the same network as SCL:
   #statVisionCmd[2] := #statAllMoveSeq = 25;
   #statTimer[4].TON(IN := (#statAllMoveSeq = 25) AND #statVisionCmd[2], PT := #VISION_DELAY_TIME);
   IF #statTimer[4].Q THEN #statAllMoveSeq := 30; END_IF;
END_REGION

REGION Network 12: All Move Seq Pos 3 [Seq 30]
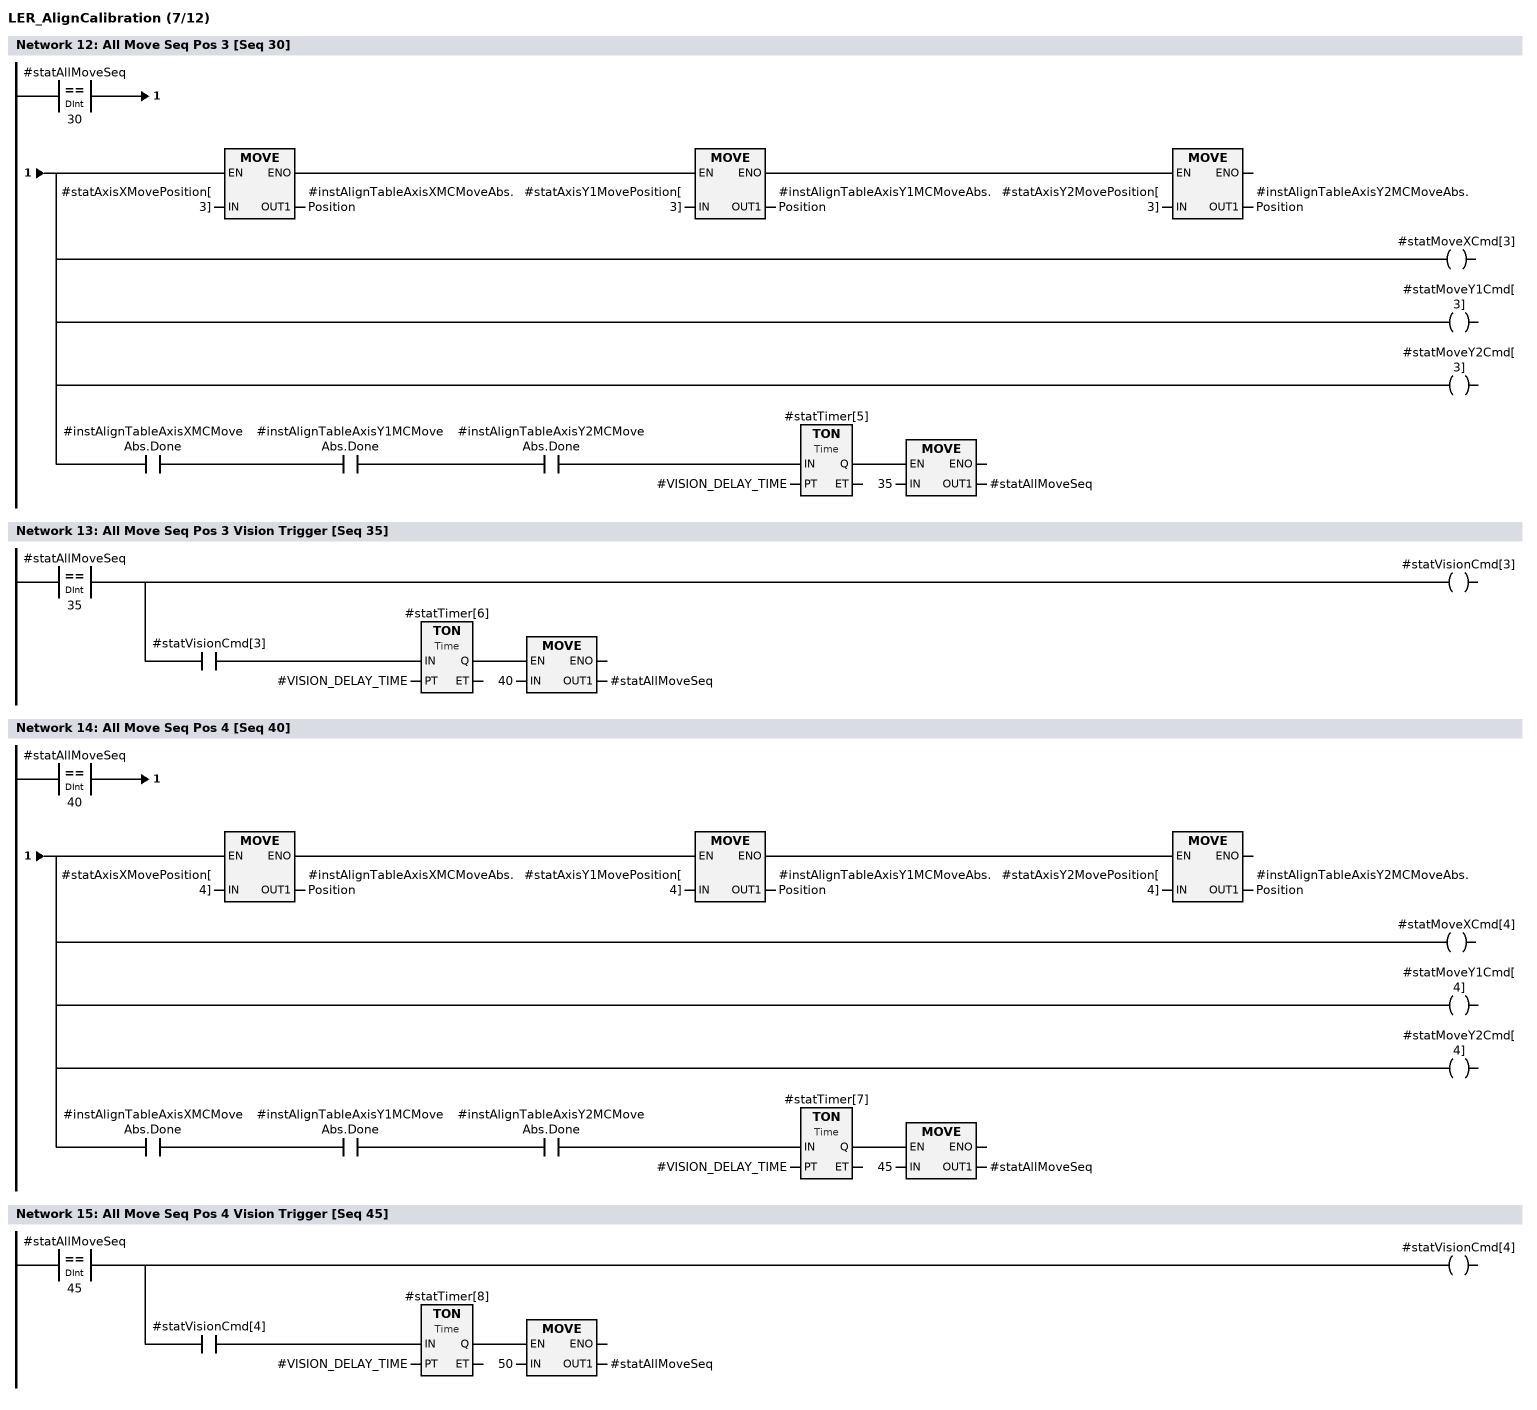
   RUNG wire#powerrail
      { S7_Templates := "SrcType := DInt" } EQ_Contact(in1 := #statAllMoveSeq, in2 := 30)
      wire#w1
      Move(in := #statAxisXMovePosition[3], out1 => #instAlignTableAxisXMCMoveAbs.Position)
      Move(in := #statAxisY1MovePosition[3], out1 => #instAlignTableAxisY1MCMoveAbs.Position)
      Move(in := #statAxisY2MovePosition[3], out1 => #instAlignTableAxisY2MCMoveAbs.Position)
   END_RUNG
   RUNG wire#w1
      Coil( #statMoveXCmd[3] )
   END_RUNG
   RUNG wire#w1
      Coil( #statMoveY1Cmd[3] )
   END_RUNG
   RUNG wire#w1
      Coil( #statMoveY2Cmd[3] )
   END_RUNG
   RUNG wire#w1
      Contact( #instAlignTableAxisXMCMoveAbs.Done )
      Contact( #instAlignTableAxisY1MCMoveAbs.Done )
      Contact( #instAlignTableAxisY2MCMoveAbs.Done )
      { S7_Templates := "time_type := Time" } #statTimer[5].TON(pt := #VISION_DELAY_TIME, et =>)
      Move(in := 35, out1 => #statAllMoveSeq)
   END_RUNG
   // the same network as SCL:
   #_w1 := #statAllMoveSeq = 30;
   IF #_w1 THEN
       #instAlignTableAxisXMCMoveAbs.Position := #statAxisXMovePosition[3];
       #instAlignTableAxisY1MCMoveAbs.Position := #statAxisY1MovePosition[3];
       #instAlignTableAxisY2MCMoveAbs.Position := #statAxisY2MovePosition[3];
   END_IF;
   #statMoveXCmd[3] := #_w1;
   #statMoveY1Cmd[3] := #_w1;
   #statMoveY2Cmd[3] := #_w1;
   #statTimer[5].TON(IN := #_w1 AND #instAlignTableAxisXMCMoveAbs.Done AND #instAlignTableAxisY1MCMoveAbs.Done AND #instAlignTableAxisY2MCMoveAbs.Done,
                     PT := #VISION_DELAY_TIME);
   IF #statTimer[5].Q THEN #statAllMoveSeq := 35; END_IF;
END_REGION

REGION Network 13: All Move Seq Pos 3 Vision Trigger [Seq 35]
   RUNG wire#powerrail
      { S7_Templates := "SrcType := DInt" } EQ_Contact(in1 := #statAllMoveSeq, in2 := 35)
      wire#w1
      Coil( #statVisionCmd[3] )
   END_RUNG
   RUNG wire#w1
      Contact( #statVisionCmd[3] )
      { S7_Templates := "time_type := Time" } #statTimer[6].TON(pt := #VISION_DELAY_TIME, et =>)
      Move(in := 40, out1 => #statAllMoveSeq)
   END_RUNG
   // the same network as SCL:
   #statVisionCmd[3] := #statAllMoveSeq = 35;
   #statTimer[6].TON(IN := (#statAllMoveSeq = 35) AND #statVisionCmd[3], PT := #VISION_DELAY_TIME);
   IF #statTimer[6].Q THEN #statAllMoveSeq := 40; END_IF;
END_REGION

REGION Network 14: All Move Seq Pos 4 [Seq 40]
   RUNG wire#powerrail
      { S7_Templates := "SrcType := DInt" } EQ_Contact(in1 := #statAllMoveSeq, in2 := 40)
      wire#w1
      Move(in := #statAxisXMovePosition[4], out1 => #instAlignTableAxisXMCMoveAbs.Position)
      Move(in := #statAxisY1MovePosition[4], out1 => #instAlignTableAxisY1MCMoveAbs.Position)
      Move(in := #statAxisY2MovePosition[4], out1 => #instAlignTableAxisY2MCMoveAbs.Position)
   END_RUNG
   RUNG wire#w1
      Coil( #statMoveXCmd[4] )
   END_RUNG
   RUNG wire#w1
      Coil( #statMoveY1Cmd[4] )
   END_RUNG
   RUNG wire#w1
      Coil( #statMoveY2Cmd[4] )
   END_RUNG
   RUNG wire#w1
      Contact( #instAlignTableAxisXMCMoveAbs.Done )
      Contact( #instAlignTableAxisY1MCMoveAbs.Done )
      Contact( #instAlignTableAxisY2MCMoveAbs.Done )
      { S7_Templates := "time_type := Time" } #statTimer[7].TON(pt := #VISION_DELAY_TIME, et =>)
      Move(in := 45, out1 => #statAllMoveSeq)
   END_RUNG
   // the same network as SCL:
   #_w1 := #statAllMoveSeq = 40;
   IF #_w1 THEN
       #instAlignTableAxisXMCMoveAbs.Position := #statAxisXMovePosition[4];
       #instAlignTableAxisY1MCMoveAbs.Position := #statAxisY1MovePosition[4];
       #instAlignTableAxisY2MCMoveAbs.Position := #statAxisY2MovePosition[4];
   END_IF;
   #statMoveXCmd[4] := #_w1;
   #statMoveY1Cmd[4] := #_w1;
   #statMoveY2Cmd[4] := #_w1;
   #statTimer[7].TON(IN := #_w1 AND #instAlignTableAxisXMCMoveAbs.Done AND #instAlignTableAxisY1MCMoveAbs.Done AND #instAlignTableAxisY2MCMoveAbs.Done,
                     PT := #VISION_DELAY_TIME);
   IF #statTimer[7].Q THEN #statAllMoveSeq := 45; END_IF;
END_REGION

REGION Network 15: All Move Seq Pos 4 Vision Trigger [Seq 45]
   RUNG wire#powerrail
      { S7_Templates := "SrcType := DInt" } EQ_Contact(in1 := #statAllMoveSeq, in2 := 45)
      wire#w1
      Coil( #statVisionCmd[4] )
   END_RUNG
   RUNG wire#w1
      Contact( #statVisionCmd[4] )
      { S7_Templates := "time_type := Time" } #statTimer[8].TON(pt := #VISION_DELAY_TIME, et =>)
      Move(in := 50, out1 => #statAllMoveSeq)
   END_RUNG
   // the same network as SCL:
   #statVisionCmd[4] := #statAllMoveSeq = 45;
   #statTimer[8].TON(IN := (#statAllMoveSeq = 45) AND #statVisionCmd[4], PT := #VISION_DELAY_TIME);
   IF #statTimer[8].Q THEN #statAllMoveSeq := 50; END_IF;
END_REGION

REGION Network 16: All Move Seq Pos 5 [Seq 50]
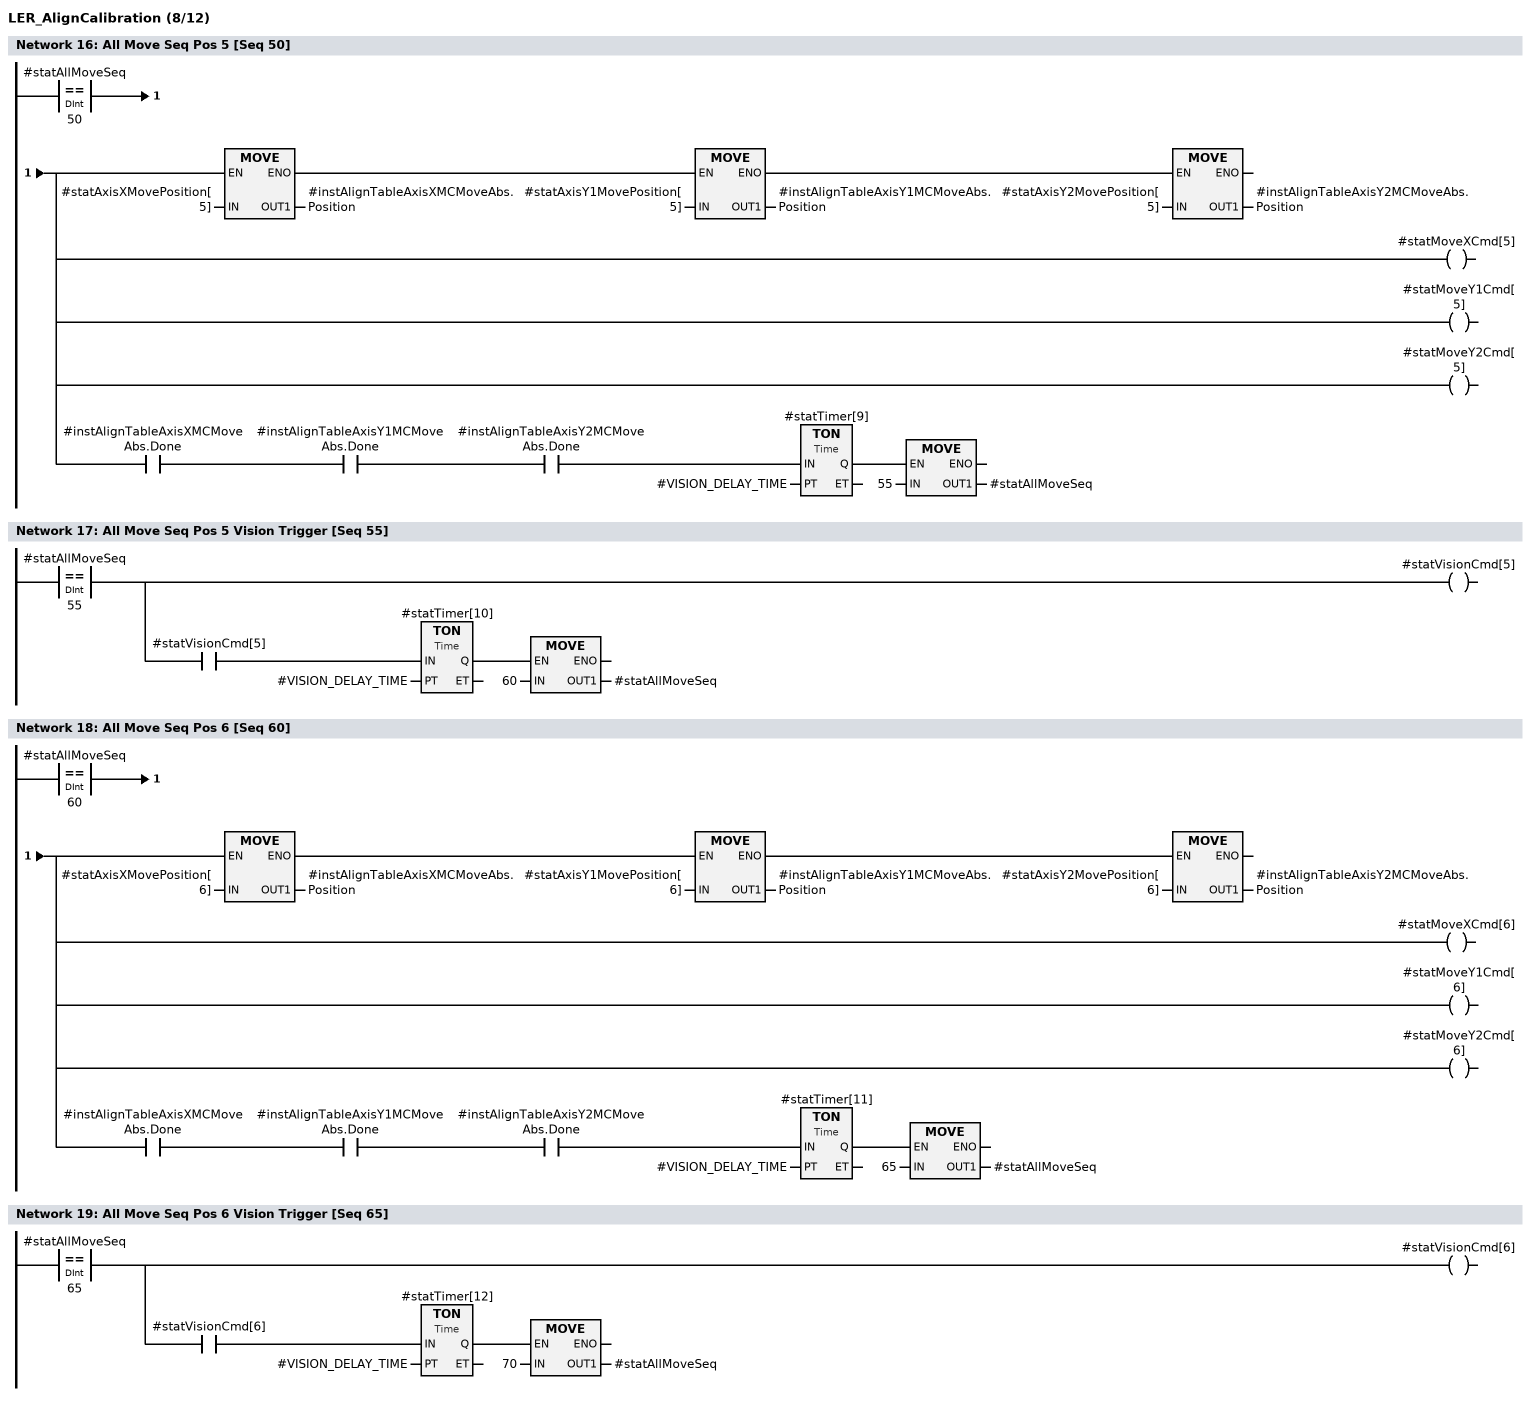
   RUNG wire#powerrail
      { S7_Templates := "SrcType := DInt" } EQ_Contact(in1 := #statAllMoveSeq, in2 := 50)
      wire#w1
      Move(in := #statAxisXMovePosition[5], out1 => #instAlignTableAxisXMCMoveAbs.Position)
      Move(in := #statAxisY1MovePosition[5], out1 => #instAlignTableAxisY1MCMoveAbs.Position)
      Move(in := #statAxisY2MovePosition[5], out1 => #instAlignTableAxisY2MCMoveAbs.Position)
   END_RUNG
   RUNG wire#w1
      Coil( #statMoveXCmd[5] )
   END_RUNG
   RUNG wire#w1
      Coil( #statMoveY1Cmd[5] )
   END_RUNG
   RUNG wire#w1
      Coil( #statMoveY2Cmd[5] )
   END_RUNG
   RUNG wire#w1
      Contact( #instAlignTableAxisXMCMoveAbs.Done )
      Contact( #instAlignTableAxisY1MCMoveAbs.Done )
      Contact( #instAlignTableAxisY2MCMoveAbs.Done )
      { S7_Templates := "time_type := Time" } #statTimer[9].TON(pt := #VISION_DELAY_TIME, et =>)
      Move(in := 55, out1 => #statAllMoveSeq)
   END_RUNG
   // the same network as SCL:
   #_w1 := #statAllMoveSeq = 50;
   IF #_w1 THEN
       #instAlignTableAxisXMCMoveAbs.Position := #statAxisXMovePosition[5];
       #instAlignTableAxisY1MCMoveAbs.Position := #statAxisY1MovePosition[5];
       #instAlignTableAxisY2MCMoveAbs.Position := #statAxisY2MovePosition[5];
   END_IF;
   #statMoveXCmd[5] := #_w1;
   #statMoveY1Cmd[5] := #_w1;
   #statMoveY2Cmd[5] := #_w1;
   #statTimer[9].TON(IN := #_w1 AND #instAlignTableAxisXMCMoveAbs.Done AND #instAlignTableAxisY1MCMoveAbs.Done AND #instAlignTableAxisY2MCMoveAbs.Done,
                     PT := #VISION_DELAY_TIME);
   IF #statTimer[9].Q THEN #statAllMoveSeq := 55; END_IF;
END_REGION

REGION Network 17: All Move Seq Pos 5 Vision Trigger [Seq 55]
   RUNG wire#powerrail
      { S7_Templates := "SrcType := DInt" } EQ_Contact(in1 := #statAllMoveSeq, in2 := 55)
      wire#w1
      Coil( #statVisionCmd[5] )
   END_RUNG
   RUNG wire#w1
      Contact( #statVisionCmd[5] )
      { S7_Templates := "time_type := Time" } #statTimer[10].TON(pt := #VISION_DELAY_TIME, et =>)
      Move(in := 60, out1 => #statAllMoveSeq)
   END_RUNG
   // the same network as SCL:
   #statVisionCmd[5] := #statAllMoveSeq = 55;
   #statTimer[10].TON(IN := (#statAllMoveSeq = 55) AND #statVisionCmd[5], PT := #VISION_DELAY_TIME);
   IF #statTimer[10].Q THEN #statAllMoveSeq := 60; END_IF;
END_REGION

REGION Network 18: All Move Seq Pos 6 [Seq 60]
   RUNG wire#powerrail
      { S7_Templates := "SrcType := DInt" } EQ_Contact(in1 := #statAllMoveSeq, in2 := 60)
      wire#w1
      Move(in := #statAxisXMovePosition[6], out1 => #instAlignTableAxisXMCMoveAbs.Position)
      Move(in := #statAxisY1MovePosition[6], out1 => #instAlignTableAxisY1MCMoveAbs.Position)
      Move(in := #statAxisY2MovePosition[6], out1 => #instAlignTableAxisY2MCMoveAbs.Position)
   END_RUNG
   RUNG wire#w1
      Coil( #statMoveXCmd[6] )
   END_RUNG
   RUNG wire#w1
      Coil( #statMoveY1Cmd[6] )
   END_RUNG
   RUNG wire#w1
      Coil( #statMoveY2Cmd[6] )
   END_RUNG
   RUNG wire#w1
      Contact( #instAlignTableAxisXMCMoveAbs.Done )
      Contact( #instAlignTableAxisY1MCMoveAbs.Done )
      Contact( #instAlignTableAxisY2MCMoveAbs.Done )
      { S7_Templates := "time_type := Time" } #statTimer[11].TON(pt := #VISION_DELAY_TIME, et =>)
      Move(in := 65, out1 => #statAllMoveSeq)
   END_RUNG
   // the same network as SCL:
   #_w1 := #statAllMoveSeq = 60;
   IF #_w1 THEN
       #instAlignTableAxisXMCMoveAbs.Position := #statAxisXMovePosition[6];
       #instAlignTableAxisY1MCMoveAbs.Position := #statAxisY1MovePosition[6];
       #instAlignTableAxisY2MCMoveAbs.Position := #statAxisY2MovePosition[6];
   END_IF;
   #statMoveXCmd[6] := #_w1;
   #statMoveY1Cmd[6] := #_w1;
   #statMoveY2Cmd[6] := #_w1;
   #statTimer[11].TON(IN := #_w1 AND #instAlignTableAxisXMCMoveAbs.Done AND #instAlignTableAxisY1MCMoveAbs.Done AND #instAlignTableAxisY2MCMoveAbs.Done,
                      PT := #VISION_DELAY_TIME);
   IF #statTimer[11].Q THEN #statAllMoveSeq := 65; END_IF;
END_REGION

REGION Network 19: All Move Seq Pos 6 Vision Trigger [Seq 65]
   RUNG wire#powerrail
      { S7_Templates := "SrcType := DInt" } EQ_Contact(in1 := #statAllMoveSeq, in2 := 65)
      wire#w1
      Coil( #statVisionCmd[6] )
   END_RUNG
   RUNG wire#w1
      Contact( #statVisionCmd[6] )
      { S7_Templates := "time_type := Time" } #statTimer[12].TON(pt := #VISION_DELAY_TIME, et =>)
      Move(in := 70, out1 => #statAllMoveSeq)
   END_RUNG
   // the same network as SCL:
   #statVisionCmd[6] := #statAllMoveSeq = 65;
   #statTimer[12].TON(IN := (#statAllMoveSeq = 65) AND #statVisionCmd[6], PT := #VISION_DELAY_TIME);
   IF #statTimer[12].Q THEN #statAllMoveSeq := 70; END_IF;
END_REGION

REGION Network 20: All Move Seq Pos 7 [Seq 70]
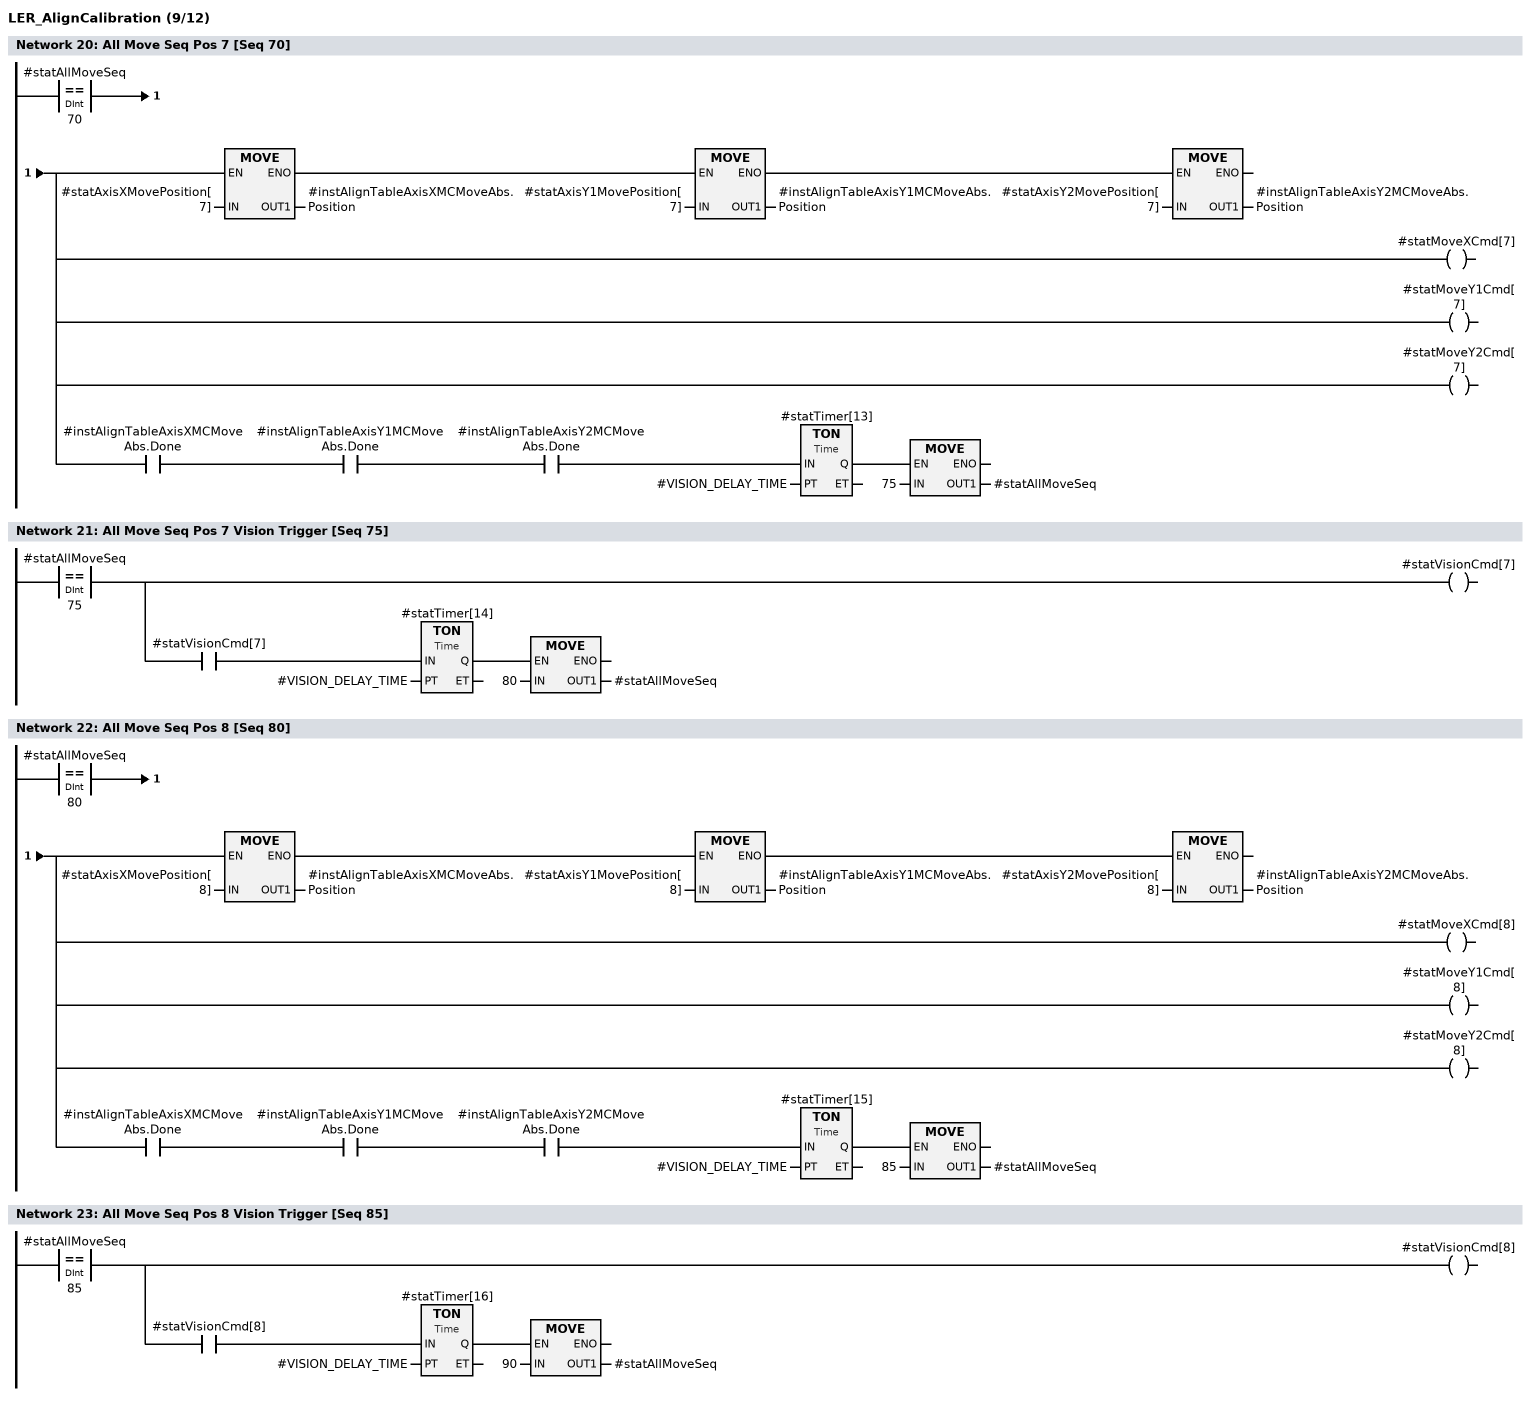
   RUNG wire#powerrail
      { S7_Templates := "SrcType := DInt" } EQ_Contact(in1 := #statAllMoveSeq, in2 := 70)
      wire#w1
      Move(in := #statAxisXMovePosition[7], out1 => #instAlignTableAxisXMCMoveAbs.Position)
      Move(in := #statAxisY1MovePosition[7], out1 => #instAlignTableAxisY1MCMoveAbs.Position)
      Move(in := #statAxisY2MovePosition[7], out1 => #instAlignTableAxisY2MCMoveAbs.Position)
   END_RUNG
   RUNG wire#w1
      Coil( #statMoveXCmd[7] )
   END_RUNG
   RUNG wire#w1
      Coil( #statMoveY1Cmd[7] )
   END_RUNG
   RUNG wire#w1
      Coil( #statMoveY2Cmd[7] )
   END_RUNG
   RUNG wire#w1
      Contact( #instAlignTableAxisXMCMoveAbs.Done )
      Contact( #instAlignTableAxisY1MCMoveAbs.Done )
      Contact( #instAlignTableAxisY2MCMoveAbs.Done )
      { S7_Templates := "time_type := Time" } #statTimer[13].TON(pt := #VISION_DELAY_TIME, et =>)
      Move(in := 75, out1 => #statAllMoveSeq)
   END_RUNG
   // the same network as SCL:
   #_w1 := #statAllMoveSeq = 70;
   IF #_w1 THEN
       #instAlignTableAxisXMCMoveAbs.Position := #statAxisXMovePosition[7];
       #instAlignTableAxisY1MCMoveAbs.Position := #statAxisY1MovePosition[7];
       #instAlignTableAxisY2MCMoveAbs.Position := #statAxisY2MovePosition[7];
   END_IF;
   #statMoveXCmd[7] := #_w1;
   #statMoveY1Cmd[7] := #_w1;
   #statMoveY2Cmd[7] := #_w1;
   #statTimer[13].TON(IN := #_w1 AND #instAlignTableAxisXMCMoveAbs.Done AND #instAlignTableAxisY1MCMoveAbs.Done AND #instAlignTableAxisY2MCMoveAbs.Done,
                      PT := #VISION_DELAY_TIME);
   IF #statTimer[13].Q THEN #statAllMoveSeq := 75; END_IF;
END_REGION

REGION Network 21: All Move Seq Pos 7 Vision Trigger [Seq 75]
   RUNG wire#powerrail
      { S7_Templates := "SrcType := DInt" } EQ_Contact(in1 := #statAllMoveSeq, in2 := 75)
      wire#w1
      Coil( #statVisionCmd[7] )
   END_RUNG
   RUNG wire#w1
      Contact( #statVisionCmd[7] )
      { S7_Templates := "time_type := Time" } #statTimer[14].TON(pt := #VISION_DELAY_TIME, et =>)
      Move(in := 80, out1 => #statAllMoveSeq)
   END_RUNG
   // the same network as SCL:
   #statVisionCmd[7] := #statAllMoveSeq = 75;
   #statTimer[14].TON(IN := (#statAllMoveSeq = 75) AND #statVisionCmd[7], PT := #VISION_DELAY_TIME);
   IF #statTimer[14].Q THEN #statAllMoveSeq := 80; END_IF;
END_REGION

REGION Network 22: All Move Seq Pos 8 [Seq 80]
   RUNG wire#powerrail
      { S7_Templates := "SrcType := DInt" } EQ_Contact(in1 := #statAllMoveSeq, in2 := 80)
      wire#w1
      Move(in := #statAxisXMovePosition[8], out1 => #instAlignTableAxisXMCMoveAbs.Position)
      Move(in := #statAxisY1MovePosition[8], out1 => #instAlignTableAxisY1MCMoveAbs.Position)
      Move(in := #statAxisY2MovePosition[8], out1 => #instAlignTableAxisY2MCMoveAbs.Position)
   END_RUNG
   RUNG wire#w1
      Coil( #statMoveXCmd[8] )
   END_RUNG
   RUNG wire#w1
      Coil( #statMoveY1Cmd[8] )
   END_RUNG
   RUNG wire#w1
      Coil( #statMoveY2Cmd[8] )
   END_RUNG
   RUNG wire#w1
      Contact( #instAlignTableAxisXMCMoveAbs.Done )
      Contact( #instAlignTableAxisY1MCMoveAbs.Done )
      Contact( #instAlignTableAxisY2MCMoveAbs.Done )
      { S7_Templates := "time_type := Time" } #statTimer[15].TON(pt := #VISION_DELAY_TIME, et =>)
      Move(in := 85, out1 => #statAllMoveSeq)
   END_RUNG
   // the same network as SCL:
   #_w1 := #statAllMoveSeq = 80;
   IF #_w1 THEN
       #instAlignTableAxisXMCMoveAbs.Position := #statAxisXMovePosition[8];
       #instAlignTableAxisY1MCMoveAbs.Position := #statAxisY1MovePosition[8];
       #instAlignTableAxisY2MCMoveAbs.Position := #statAxisY2MovePosition[8];
   END_IF;
   #statMoveXCmd[8] := #_w1;
   #statMoveY1Cmd[8] := #_w1;
   #statMoveY2Cmd[8] := #_w1;
   #statTimer[15].TON(IN := #_w1 AND #instAlignTableAxisXMCMoveAbs.Done AND #instAlignTableAxisY1MCMoveAbs.Done AND #instAlignTableAxisY2MCMoveAbs.Done,
                      PT := #VISION_DELAY_TIME);
   IF #statTimer[15].Q THEN #statAllMoveSeq := 85; END_IF;
END_REGION

REGION Network 23: All Move Seq Pos 8 Vision Trigger [Seq 85]
   RUNG wire#powerrail
      { S7_Templates := "SrcType := DInt" } EQ_Contact(in1 := #statAllMoveSeq, in2 := 85)
      wire#w1
      Coil( #statVisionCmd[8] )
   END_RUNG
   RUNG wire#w1
      Contact( #statVisionCmd[8] )
      { S7_Templates := "time_type := Time" } #statTimer[16].TON(pt := #VISION_DELAY_TIME, et =>)
      Move(in := 90, out1 => #statAllMoveSeq)
   END_RUNG
   // the same network as SCL:
   #statVisionCmd[8] := #statAllMoveSeq = 85;
   #statTimer[16].TON(IN := (#statAllMoveSeq = 85) AND #statVisionCmd[8], PT := #VISION_DELAY_TIME);
   IF #statTimer[16].Q THEN #statAllMoveSeq := 90; END_IF;
END_REGION

REGION Network 24: All Move Seq Pos 9 [Seq 90]
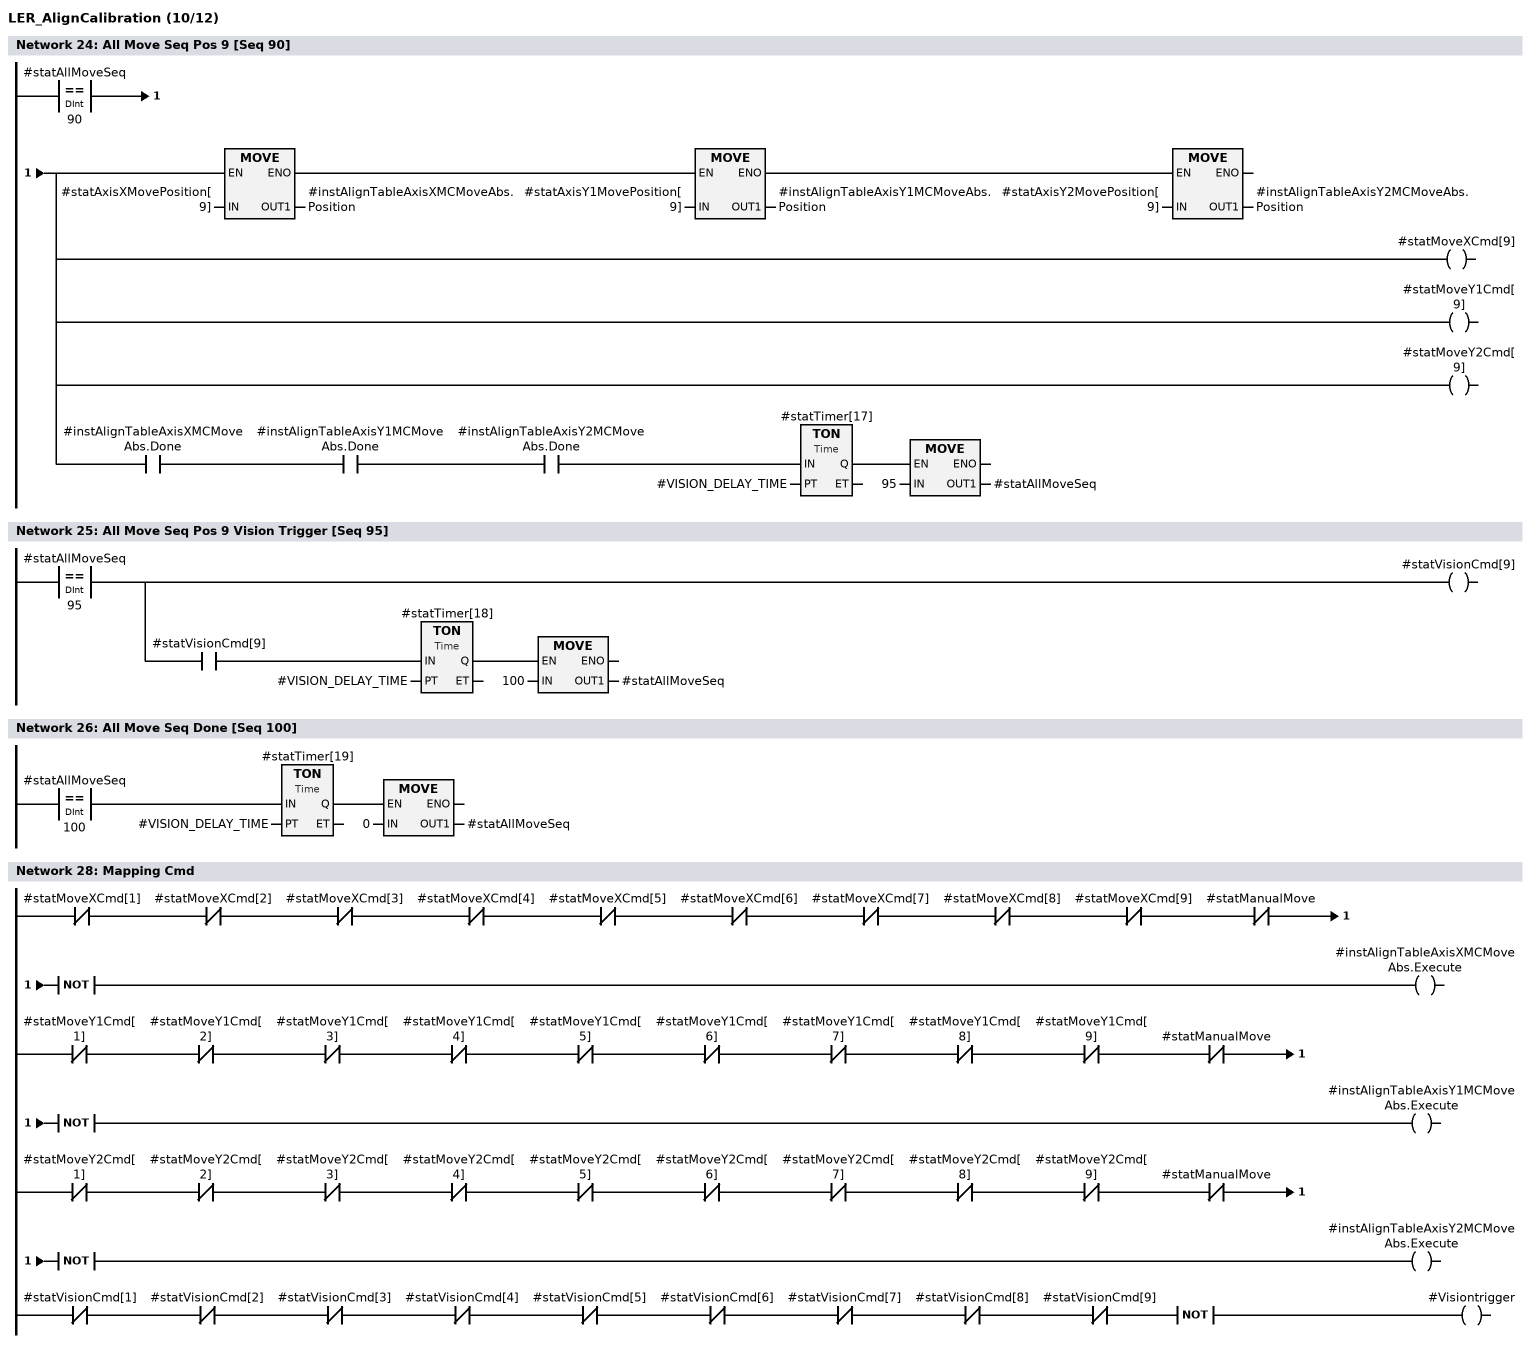
   RUNG wire#powerrail
      { S7_Templates := "SrcType := DInt" } EQ_Contact(in1 := #statAllMoveSeq, in2 := 90)
      wire#w1
      Move(in := #statAxisXMovePosition[9], out1 => #instAlignTableAxisXMCMoveAbs.Position)
      Move(in := #statAxisY1MovePosition[9], out1 => #instAlignTableAxisY1MCMoveAbs.Position)
      Move(in := #statAxisY2MovePosition[9], out1 => #instAlignTableAxisY2MCMoveAbs.Position)
   END_RUNG
   RUNG wire#w1
      Coil( #statMoveXCmd[9] )
   END_RUNG
   RUNG wire#w1
      Coil( #statMoveY1Cmd[9] )
   END_RUNG
   RUNG wire#w1
      Coil( #statMoveY2Cmd[9] )
   END_RUNG
   RUNG wire#w1
      Contact( #instAlignTableAxisXMCMoveAbs.Done )
      Contact( #instAlignTableAxisY1MCMoveAbs.Done )
      Contact( #instAlignTableAxisY2MCMoveAbs.Done )
      { S7_Templates := "time_type := Time" } #statTimer[17].TON(pt := #VISION_DELAY_TIME, et =>)
      Move(in := 95, out1 => #statAllMoveSeq)
   END_RUNG
   // the same network as SCL:
   #_w1 := #statAllMoveSeq = 90;
   IF #_w1 THEN
       #instAlignTableAxisXMCMoveAbs.Position := #statAxisXMovePosition[9];
       #instAlignTableAxisY1MCMoveAbs.Position := #statAxisY1MovePosition[9];
       #instAlignTableAxisY2MCMoveAbs.Position := #statAxisY2MovePosition[9];
   END_IF;
   #statMoveXCmd[9] := #_w1;
   #statMoveY1Cmd[9] := #_w1;
   #statMoveY2Cmd[9] := #_w1;
   #statTimer[17].TON(IN := #_w1 AND #instAlignTableAxisXMCMoveAbs.Done AND #instAlignTableAxisY1MCMoveAbs.Done AND #instAlignTableAxisY2MCMoveAbs.Done,
                      PT := #VISION_DELAY_TIME);
   IF #statTimer[17].Q THEN #statAllMoveSeq := 95; END_IF;
END_REGION

REGION Network 25: All Move Seq Pos 9 Vision Trigger [Seq 95]
   RUNG wire#powerrail
      { S7_Templates := "SrcType := DInt" } EQ_Contact(in1 := #statAllMoveSeq, in2 := 95)
      wire#w1
      Coil( #statVisionCmd[9] )
   END_RUNG
   RUNG wire#w1
      Contact( #statVisionCmd[9] )
      { S7_Templates := "time_type := Time" } #statTimer[18].TON(pt := #VISION_DELAY_TIME, et =>)
      Move(in := 100, out1 => #statAllMoveSeq)
   END_RUNG
   // the same network as SCL:
   #statVisionCmd[9] := #statAllMoveSeq = 95;
   #statTimer[18].TON(IN := (#statAllMoveSeq = 95) AND #statVisionCmd[9], PT := #VISION_DELAY_TIME);
   IF #statTimer[18].Q THEN #statAllMoveSeq := 100; END_IF;
END_REGION

REGION Network 26: All Move Seq Done [Seq 100]
   RUNG wire#powerrail
      { S7_Templates := "SrcType := DInt" } EQ_Contact(in1 := #statAllMoveSeq, in2 := 100)
      { S7_Templates := "time_type := Time" } #statTimer[19].TON(pt := #VISION_DELAY_TIME, et =>)
      Move(in := 0, out1 => #statAllMoveSeq)
   END_RUNG
   // the same network as SCL:
   #statTimer[19].TON(IN := #statAllMoveSeq = 100, PT := #VISION_DELAY_TIME);
   IF #statTimer[19].Q THEN #statAllMoveSeq := 0; END_IF;
END_REGION

REGION Network 27: === Sequence End ===
END_REGION

REGION Network 28: Mapping Cmd
   RUNG wire#powerrail
      I_Contact( #statMoveXCmd[1] )
      I_Contact( #statMoveXCmd[2] )
      I_Contact( #statMoveXCmd[3] )
      I_Contact( #statMoveXCmd[4] )
      I_Contact( #statMoveXCmd[5] )
      I_Contact( #statMoveXCmd[6] )
      I_Contact( #statMoveXCmd[7] )
      I_Contact( #statMoveXCmd[8] )
      I_Contact( #statMoveXCmd[9] )
      I_Contact( #statManualMove )
      Not()
      Coil( #instAlignTableAxisXMCMoveAbs.Execute )
   END_RUNG
   RUNG wire#powerrail
      I_Contact( #statMoveY1Cmd[1] )
      I_Contact( #statMoveY1Cmd[2] )
      I_Contact( #statMoveY1Cmd[3] )
      I_Contact( #statMoveY1Cmd[4] )
      I_Contact( #statMoveY1Cmd[5] )
      I_Contact( #statMoveY1Cmd[6] )
      I_Contact( #statMoveY1Cmd[7] )
      I_Contact( #statMoveY1Cmd[8] )
      I_Contact( #statMoveY1Cmd[9] )
      I_Contact( #statManualMove )
      Not()
      Coil( #instAlignTableAxisY1MCMoveAbs.Execute )
   END_RUNG
   RUNG wire#powerrail
      I_Contact( #statMoveY2Cmd[1] )
      I_Contact( #statMoveY2Cmd[2] )
      I_Contact( #statMoveY2Cmd[3] )
      I_Contact( #statMoveY2Cmd[4] )
      I_Contact( #statMoveY2Cmd[5] )
      I_Contact( #statMoveY2Cmd[6] )
      I_Contact( #statMoveY2Cmd[7] )
      I_Contact( #statMoveY2Cmd[8] )
      I_Contact( #statMoveY2Cmd[9] )
      I_Contact( #statManualMove )
      Not()
      Coil( #instAlignTableAxisY2MCMoveAbs.Execute )
   END_RUNG
   RUNG wire#powerrail
      I_Contact( #statVisionCmd[1] )
      I_Contact( #statVisionCmd[2] )
      I_Contact( #statVisionCmd[3] )
      I_Contact( #statVisionCmd[4] )
      I_Contact( #statVisionCmd[5] )
      I_Contact( #statVisionCmd[6] )
      I_Contact( #statVisionCmd[7] )
      I_Contact( #statVisionCmd[8] )
      I_Contact( #statVisionCmd[9] )
      Not()
      Coil( #Visiontrigger )
   END_RUNG
   // the same network as SCL:
   #instAlignTableAxisXMCMoveAbs.Execute := NOT (NOT #statMoveXCmd[1] AND NOT #statMoveXCmd[2] AND NOT #statMoveXCmd[3] AND NOT #statMoveXCmd[4] AND NOT #statMoveXCmd[5] AND NOT #statMoveXCmd[6] AND NOT #statMoveXCmd[7] AND NOT #statMoveXCmd[8] AND NOT #statMoveXCmd[9] AND NOT #statManualMove);
   #instAlignTableAxisY1MCMoveAbs.Execute := NOT (NOT #statMoveY1Cmd[1] AND NOT #statMoveY1Cmd[2] AND NOT #statMoveY1Cmd[3] AND NOT #statMoveY1Cmd[4] AND NOT #statMoveY1Cmd[5] AND NOT #statMoveY1Cmd[6] AND NOT #statMoveY1Cmd[7] AND NOT #statMoveY1Cmd[8] AND NOT #statMoveY1Cmd[9] AND NOT #statManualMove);
   #instAlignTableAxisY2MCMoveAbs.Execute := NOT (NOT #statMoveY2Cmd[1] AND NOT #statMoveY2Cmd[2] AND NOT #statMoveY2Cmd[3] AND NOT #statMoveY2Cmd[4] AND NOT #statMoveY2Cmd[5] AND NOT #statMoveY2Cmd[6] AND NOT #statMoveY2Cmd[7] AND NOT #statMoveY2Cmd[8] AND NOT #statMoveY2Cmd[9] AND NOT #statManualMove);
   #Visiontrigger := NOT (NOT #statVisionCmd[1] AND NOT #statVisionCmd[2] AND NOT #statVisionCmd[3] AND NOT #statVisionCmd[4] AND NOT #statVisionCmd[5] AND NOT #statVisionCmd[6] AND NOT #statVisionCmd[7] AND NOT #statVisionCmd[8] AND NOT #statVisionCmd[9]);
END_REGION

REGION Network 29: Call Instance
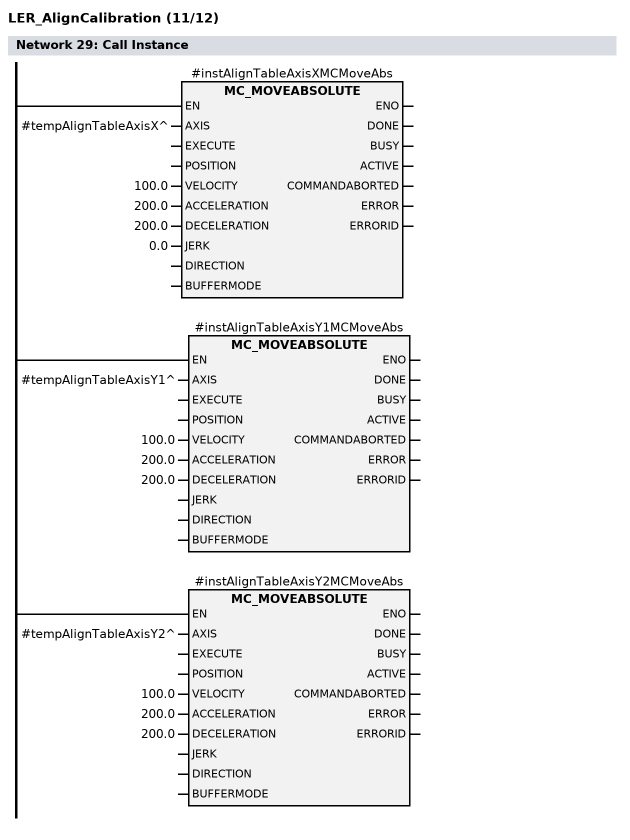
   RUNG wire#powerrail
      #instAlignTableAxisXMCMoveAbs.MC_MOVEABSOLUTE(Axis := #tempAlignTableAxisX^, Execute :=, Position :=, Velocity := 100.0, Acceleration := 200.0, Deceleration := 200.0, Jerk := 0.0, Direction :=, BufferMode :=, Done =>, Busy =>, Active =>, CommandAborted =>, Error =>, ErrorId =>)
   END_RUNG
   RUNG wire#powerrail
      #instAlignTableAxisY1MCMoveAbs.MC_MOVEABSOLUTE(Axis := #tempAlignTableAxisY1^, Execute :=, Position :=, Velocity := 100.0, Acceleration := 200.0, Deceleration := 200.0, Jerk :=, Direction :=, BufferMode :=, Done =>, Busy =>, Active =>, CommandAborted =>, Error =>, ErrorId =>)
   END_RUNG
   RUNG wire#powerrail
      #instAlignTableAxisY2MCMoveAbs.MC_MOVEABSOLUTE(Axis := #tempAlignTableAxisY2^, Execute :=, Position :=, Velocity := 100.0, Acceleration := 200.0, Deceleration := 200.0, Jerk :=, Direction :=, BufferMode :=, Done =>, Busy =>, Active =>, CommandAborted =>, Error =>, ErrorId =>)
   END_RUNG
   // the same network as SCL:
   #instAlignTableAxisXMCMoveAbs(Axis := #tempAlignTableAxisX^,   // MC_MOVEABSOLUTE
                           Velocity := 100.0,
                           Acceleration := 200.0,
                           Deceleration := 200.0,
                           Jerk := 0.0);
   #instAlignTableAxisY1MCMoveAbs(Axis := #tempAlignTableAxisY1^,   // MC_MOVEABSOLUTE
                           Velocity := 100.0,
                           Acceleration := 200.0,
                           Deceleration := 200.0);
   #instAlignTableAxisY2MCMoveAbs(Axis := #tempAlignTableAxisY2^,   // MC_MOVEABSOLUTE
                           Velocity := 100.0,
                           Acceleration := 200.0,
                           Deceleration := 200.0);
END_REGION

REGION Network 30: Mapping Output
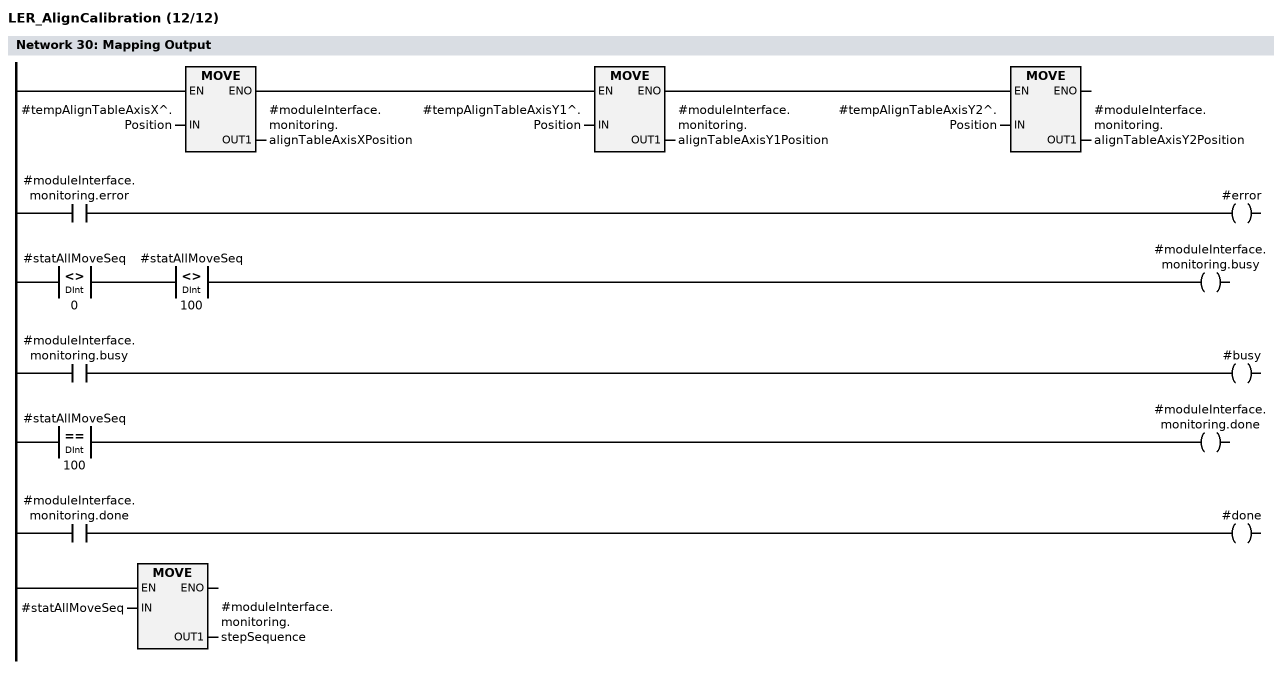
   RUNG wire#powerrail
      Move(in := #tempAlignTableAxisX^.Position, out1 => #moduleInterface.monitoring.alignTableAxisXPosition)
      Move(in := #tempAlignTableAxisY1^.Position, out1 => #moduleInterface.monitoring.alignTableAxisY1Position)
      Move(in := #tempAlignTableAxisY2^.Position, out1 => #moduleInterface.monitoring.alignTableAxisY2Position)
   END_RUNG
   RUNG wire#powerrail
      Contact( #moduleInterface.monitoring.error )
      Coil( #error )
   END_RUNG
   RUNG wire#powerrail
      { S7_Templates := "SrcType := DInt" } NE_Contact(in1 := #statAllMoveSeq, in2 := 0)
      { S7_Templates := "SrcType := DInt" } NE_Contact(in1 := #statAllMoveSeq, in2 := 100)
      Coil( #moduleInterface.monitoring.busy )
   END_RUNG
   RUNG wire#powerrail
      Contact( #moduleInterface.monitoring.busy )
      Coil( #busy )
   END_RUNG
   RUNG wire#powerrail
      { S7_Templates := "SrcType := DInt" } EQ_Contact(in1 := #statAllMoveSeq, in2 := 100)
      Coil( #moduleInterface.monitoring.done )
   END_RUNG
   RUNG wire#powerrail
      Contact( #moduleInterface.monitoring.done )
      Coil( #done )
   END_RUNG
   RUNG wire#powerrail
      Move(in := #statAllMoveSeq, out1 => #moduleInterface.monitoring.stepSequence)
   END_RUNG
   // the same network as SCL:
   #moduleInterface.monitoring.alignTableAxisXPosition := #tempAlignTableAxisX^.Position;
   #moduleInterface.monitoring.alignTableAxisY1Position := #tempAlignTableAxisY1^.Position;
   #moduleInterface.monitoring.alignTableAxisY2Position := #tempAlignTableAxisY2^.Position;
   #error := #moduleInterface.monitoring.error;
   #moduleInterface.monitoring.busy := (#statAllMoveSeq <> 0) AND (#statAllMoveSeq <> 100);
   #busy := #moduleInterface.monitoring.busy;
   #moduleInterface.monitoring.done := #statAllMoveSeq = 100;
   #done := #moduleInterface.monitoring.done;
   #moduleInterface.monitoring.stepSequence := #statAllMoveSeq;
END_REGION
END_FUNCTION_BLOCK
